		IF CalcolaFormingRT[IdxLista] AND NOT CalcolaFormingRT2[IdxLista] AND ActualPickingListFromHMI[IdxLista].State = 1   THEN //###############################  If  Principal calculos formaciones bendel y cabaleta
				 		//Para quitar
		Control1 := control1 +1 ;
			IF TFCalcoloFormaturaRT[IdxLista].CalcolaFormaturaDone THEN
				CalcolaFormaturaTrig2 := TRUE;	  
			END_IF
			IF NOT CalcolaFormaturaTrig2 AND NOT Formacion_bandelCalOk[idxForm]  THEN//11111111111111111
			///////////////////////////
				//CalcolaFormaturaTrig2 := TRUE;
				TFCalcoloFormaturaRT[IdxLista].PulisciMemoria 	:= TRUE;
				IF TFCalcoloFormaturaRT[IdxLista].PulisciMemoriaDone THEN		
					FOR i:= 1 TO MAXFORMINGSLAB DO
						IF i <= 40 THEN
						//IF i <= HMI_Forming_NumeroElementiDaDepositare THEN
							TFCalcoloFormaturaRT[IdxLista].TipoElementoDep[i] := LASTRA;//Settiamo tutte lastre!!
						ELSE
							TFCalcoloFormaturaRT[IdxLista].TipoElementoDep[i] := TERMINATORE;//Settiamo il resto come terminatore
						END_IF
					END_FOR
					TFCalcoloFormaturaRT[IdxLista].Materiale[e_Tipo_Elemento_Da_Lavorare.LASTRA].XDim		:= RequestPickingListFromHMI[IdxLista].SlabDimension.XDim; 
					TFCalcoloFormaturaRT[IdxLista].Materiale[e_Tipo_Elemento_Da_Lavorare.LASTRA].YDim		:= RequestPickingListFromHMI[IdxLista].SlabDimension.YDim; 
					TFCalcoloFormaturaRT[IdxLista].Materiale[e_Tipo_Elemento_Da_Lavorare.LASTRA].ZDim		:= RequestPickingListFromHMI[IdxLista].SlabDimension.ZDim; 
					TFCalcoloFormaturaRT[IdxLista].Supporto.Code											:= RequestPickingListFromHMI[IdxLista].SupportVertBundle.Code;
					TFCalcoloFormaturaRT[IdxLista].Supporto.XDim											:= RequestPickingListFromHMI[IdxLista].SupportVertBundle.XDim;
					TFCalcoloFormaturaRT[IdxLista].Supporto.YDim											:= RequestPickingListFromHMI[IdxLista].SupportVertBundle.YDim*2;
					TFCalcoloFormaturaRT[IdxLista].Supporto.ZDim				:= RequestPickingListFromHMI[IdxLista].SupportVertBundle.ZDim;
					TFCalcoloFormaturaRT[IdxLista].Supporto.TipoPianoAppoggio 	:= 1;
					TFCalcoloFormaturaRT[IdxLista].Supporto.AltezzaDenteRitenuta:= 15;
					TFCalcoloFormaturaRT[IdxLista].Supporto.ZDim_Ext1        	:= TFCalcoloFormaturaRT[IdxLista].Supporto.ZDim + TFCalcoloFormaturaRT[IdxLista].Supporto.AltezzaDenteRitenuta;
					TFCalcoloFormaturaRT[IdxLista].Supporto.DimBaseUtile		:= RequestPickingListFromHMI[IdxLista].SupportVertBundle.DimBaseUtile;
					TFCalcoloFormaturaRT[IdxLista].Supporto.DimVertice 			:= RequestPickingListFromHMI[IdxLista].SupportVertBundle.DimVertice*2;
					TFCalcoloFormaturaRT[IdxLista].Supporto.HMAX 				:= RequestPickingListFromHMI[IdxLista].SupportVertBundle.HMAX;
					TFCalcoloFormaturaRT[IdxLista].Supporto.Tipologia 			:= BUNDLE;
					TFCalcoloFormaturaRT[IdxLista].Supporto.LatoDeposito 		:= 180;
					TFCalcoloFormaturaRT[IdxLista].TipoOrdinamento				:= 4;	//Ordinamento di deposito, prima un lato poi l'altro
					TFCalcoloFormaturaRT[IdxLista].CalcolaFormatura 			:= TRUE;//Lancio esecuzione dei calcoli
					MEMSET(ADR(FormaturaBundleRT[IdxLista]),0,SIZEOF(FormaturaBundleRT[IdxLista]));	//Pulisco la memoria di destinazione
					TFCalcoloFormaturaRT[IdxLista].PulisciMemoria := FALSE;
				END_IF
			ELSIF (TFCalcoloFormaturaRT[IdxLista].CalcolaFormaturaDone OR TFCalcoloFormaturaRT[IdxLista].Errore > 0) AND CalcolaFormaturaTrig2 THEN
				CalcolaFormaturaTrig2 := FALSE;
				TFCalcoloFormaturaRT[IdxLista].CalcolaFormatura := FALSE;
				TFFormacionBandelCalculada := TFCalcoloFormaturaRT[IdxLista]; 
				FormaturaBundleRT[IdxLista] := TFCalcoloFormaturaRT[IdxLista].FormingSlab;
				IF TFCalcoloFormaturaRT[IdxLista].Errore = 0 THEN
					CalcolaFormaturaTrig2 			:= FALSE;
					CalcolaFormingRT[IdxLista] 		:= FALSE;
					CalcolaFormingRT2[IdxLista]		:= TRUE;
					Formacion_bandelCalOk[idxForm] 			:= TRUE ;
				ELSE
					CalcolaFormingRT[IdxLista] 		:= TRUE;
					CalcolaFormaturaTrig2 			:= FALSE;
				END_IF
			END_IF
		//##############################Inicio##############################################		 
		//#########################Calculo cavaleta##########################################
		ELSIF CalcolaFormingRT2[IdxLista] AND NOT CalcolaFormingRT[IdxLista] AND ActualPickingListFromHMI[IdxLista].State = 1  THEN 
			IF NOT CalcolaFormaturaTrig2 AND NOT Formacion_FrameCalOk[idxForm] THEN
			///////////////////////////
				TFCalcoloFormaturaRT[IdxLista].PulisciMemoria 	:= TRUE;	  
				
					
				//TFCalcoloFormaturaRT[IdxLista].PulisciMemoria 	:= TRUE;
				IF TFCalcoloFormaturaRT[IdxLista].PulisciMemoriaDone THEN
					CalcolaFormaturaTrig2 := TRUE;		
					FOR i:= 1 TO MAXFORMINGSLAB DO
						//IF i <= 10  THEN
						IF i <= 40 THEN
						//IF i <= HMI_Forming_NumeroElementiDaDepositare  THEN
							TFCalcoloFormaturaRT[IdxLista].TipoElementoDep[i] := LASTRA;//Settiamo tutte lastre!!
						ELSE
							TFCalcoloFormaturaRT[IdxLista].TipoElementoDep[i] := TERMINATORE;//Settiamo il resto come terminatore
						END_IF
					END_FOR
					TFCalcoloFormaturaRT[IdxLista].Materiale[e_Tipo_Elemento_Da_Lavorare.LASTRA].XDim		:= RequestPickingListFromHMI[IdxLista].SlabDimension.XDim; 
					TFCalcoloFormaturaRT[IdxLista].Materiale[e_Tipo_Elemento_Da_Lavorare.LASTRA].YDim		:= RequestPickingListFromHMI[IdxLista].SlabDimension.YDim; 
					TFCalcoloFormaturaRT[IdxLista].Materiale[e_Tipo_Elemento_Da_Lavorare.LASTRA].ZDim		:= RequestPickingListFromHMI[IdxLista].SlabDimension.ZDim; 
					TFCalcoloFormaturaRT[IdxLista].HabiCalTodasCordenadas := true ;
					TFCalcoloFormaturaRT[IdxLista].Supporto.Code											:= RequestPickingListFromHMI[IdxLista].SupportVertCav.Code;
					TFCalcoloFormaturaRT[IdxLista].Supporto.XDim											:= RequestPickingListFromHMI[IdxLista].SupportVertCav.XDim;
					TFCalcoloFormaturaRT[IdxLista].Supporto.YDim											:= RequestPickingListFromHMI[IdxLista].SupportVertCav.YDim(**2*);
					TFCalcoloFormaturaRT[IdxLista].Supporto.ZDim				:= RequestPickingListFromHMI[IdxLista].SupportVertCav.ZDim;
					TFCalcoloFormaturaRT[IdxLista].Supporto.TipoPianoAppoggio 	:= 1;
					TFCalcoloFormaturaRT[IdxLista].Supporto.AltezzaDenteRitenuta:= 13;
					TFCalcoloFormaturaRT[IdxLista].Supporto.ZDim_Ext1        	:= TFCalcoloFormaturaRT[IdxLista].Supporto.ZDim + TFCalcoloFormaturaRT[IdxLista].Supporto.AltezzaDenteRitenuta;
					TFCalcoloFormaturaRT[IdxLista].Supporto.DimBaseUtile		:= RequestPickingListFromHMI[IdxLista].SupportVertCav.DimBaseUtile;
					TFCalcoloFormaturaRT[IdxLista].Supporto.DimVertice 			:= RequestPickingListFromHMI[IdxLista].SupportVertCav.DimVertice(**2*);
					TFCalcoloFormaturaRT[IdxLista].Supporto.HMAX 				:= RequestPickingListFromHMI[IdxLista].SupportVertCav.HMAX;
					TFCalcoloFormaturaRT[IdxLista].Supporto.Tipologia 			:= CAVALLETTO;
					TFCalcoloFormaturaRT[IdxLista].Supporto.LatoDeposito 		:= 0;
					TFCalcoloFormaturaRT[IdxLista].TipoOrdinamento				:= 1;	//Ordinamento di deposito, prima un lato poi l'altro
					TFCalcoloFormaturaRT[IdxLista].CalcolaFormatura 			:= TRUE;//Lancio esecuzione dei calcoli
					MEMSET(ADR(FormaturaAFRAMERT[IdxLista]),0,SIZEOF(FormaturaAFRAMERT[IdxLista]));	//Pulisco la memoria di destinazione
					TFCalcoloFormaturaRT[IdxLista].PulisciMemoria := FALSE;
				END_IF
			ELSIF (TFCalcoloFormaturaRT[IdxLista].CalcolaFormaturaDone OR TFCalcoloFormaturaRT[IdxLista].Errore > 0) AND CalcolaFormaturaTrig2 THEN
				CalcolaFormaturaTrig2 		:= FALSE;
				TFCalcoloFormaturaRT[IdxLista].CalcolaFormatura := FALSE;
				TFFormacionCavalleteCalculada := TFCalcoloFormaturaRT[IdxLista] ;
				FormaturaAFRAMERT[IdxLista] := TFCalcoloFormaturaRT[IdxLista].FormingSlab;
				
				//CalcolaFormingRT[IdxLista] := TRUE ; // modificacion probar
				IF TFCalcoloFormaturaRT[IdxLista].Errore = 0 THEN
					CalcolaFormaturaTrig2 		:= FALSE;
					CalcolaFormingRT[IdxLista] 	:= TRUE;
					CalcolaFormingRT2[IdxLista]	:= FALSE;
					Formacion_FrameCalOk[idxForm] 		:= TRUE ;
				ELSE
					//CalcolaFormingRT[IdxLista] := TRUE; // original	  
					CalcolaFormingRT2[IdxLista] := TRUE;
				//##############################Fin ##############################################		 
				//#########################Calculo cavaleta##########################################
				END_IF
			END_IF
				  
		END_IF //###############################  If  Principal calculos formaciones bendel y cabaleta
	
	TFCalcoloFormaturaRT[IdxLista]();
END_FOR	 
	 

	HMI_WorkAreaDataPicking_1_8 := ActualPickingListFromHMI[1].State >= 1;//Ordine postazioni 1..8 in lavoro
		 
	HMI_WorkAreaDataPicking_1_4 := (ActualPickingListFromHMI[2].State >= 1);//Ordine postazioni 1..4 in lavoro
	HMI_WorkAreaDataPicking_5_8 := (ActualPickingListFromHMI[3].State >= 1);//Ordine postazioni 5..8 in lavoro

//FOR IdxLista := 1 TO 3 DO
//	CASE IdxLista OF	 
//		1: Iforstart := 1; Iforend := MAXAREAPRESENT;
//		2: Iforstart := 1; Iforend := 4;
//		3: Iforstart := 5; Iforend := MAXAREAPRESENT;
//	END_CASE		 		   
//	FOR i:= Iforstart TO Iforend DO	
//		IF NumeroPezziPresentiPostazioneStart[i] = 0 AND WorkAreaState[i].P > 1 THEN
//			NumeroPezziPresentiPostazioneStart[i] := TO_UINT(WorkAreaState[i].P);
//		END_IF
//	
//		IF NOT HMI_WorkAreaDataPicking[i].Destinazione THEN
//			IF HMI_WorkAreaDataPicking[i].NumElementiDaLavorare > 0 THEN
//				//IF HMI_WorkAreaDataPicking[i].NumElementiDaLavorare >= TO_UINT(WorkAreaState[i].P)-1 THEN
//				//	HMI_NumeroLastreRimanentiOrdineAttuale[i] := HMI_WorkAreaDataPicking[i].NumElementiDaLavorare - TO_UINT(WorkAreaState[i].P);
//				//ELSE
//				//	HMI_NumeroLastreRimanentiOrdineAttuale[i] := 0;
//				//END_IF
//				IF HMI_WorkAreaDataPicking[i].NumElementiDaLavorare - (TO_UINT(WorkAreaState[i].P) - NumeroPezziPresentiPostazioneStart[i]) > 0 THEN
//					HMI_NumeroLastreRimanentiOrdineAttuale[i] := MIN(HMI_WorkAreaDataPicking[i].NumElementiDaLavorare,HMI_WorkAreaDataPicking[i].NumElementiDaLavorare - 
//																(NumeroPezziPresentiPostazioneStart[i] - TO_UINT(WorkAreaState[i].P)));
//				ELSE
//					HMI_NumeroLastreRimanentiOrdineAttuale[i] := 0;
//				END_IF
//			ELSE
//				HMI_NumeroLastreRimanentiOrdineAttuale[i] := 0;
//			END_IF
//		ELSE
//			IF NumeroPezziPresentiPostazioneStart[i] <= (TO_UINT(WorkAreaState[i].P)) AND NumeroPezziPresentiPostazioneStart[i]>0 THEN
//				HMI_NumeroLastreRimanentiOrdineAttuale[i] := TO_UINT(WorkAreaState[i].P) - NumeroPezziPresentiPostazioneStart[i]+1;
//			ELSE
//				HMI_NumeroLastreRimanentiOrdineAttuale[i] := 0;
//			END_IF
//		END_IF
//		IF (WorkAreaProductionList[i].Stato = e_Stato_ListaDiProduzione.LISTA_PROD_IN_ESECUZIONE OR WorkAreaProductionList[i].Stato = e_Stato_ListaDiProduzione.LISTA_PROD_ESEGUITA) AND WorkAreaState[i].P > 1 THEN
//			HMI_NumeroLastreDepOrdineAttuale[IdxLista] := TO_UINT(WorkAreaState[i].P-1);
//			IF NumeroPezziPresentiPostazioneStart[i] < (TO_UINT(WorkAreaState[i].P)) AND NumeroPezziPresentiPostazioneStart[i]>0 THEN
//				HMI_NumeroLastreDepOrdineAttuale[IdxLista] := TO_UINT(WorkAreaState[i].P) - NumeroPezziPresentiPostazioneStart[i] +1;
//			ELSE
//				HMI_NumeroLastreDepOrdineAttuale[IdxLista] := 0;
//			END_IF
//		END_IF	
//	END_FOR		  
//END_FOR			   
					
						 
							  
								   
{endregion}
END_ACTION

ACTION _11_CalcolaListaProduzioneNew:
{region "Gestione zona GLOBALE - Postazioni da 1 a 8"}


//#############################################################################################################



	  
	  

FOR LoopLista := 1 TO 3 DO
	IdxLista := LoopLista;		 
	 // IdxLista := 2;		  
	CASE IdxLista OF	 
		1: Iforstart := 1; Iforend := MAXAREAPRESENT;
		2: Iforstart := 1; Iforend := 4;
		3: Iforstart := 5; Iforend := MAXAREAPRESENT;
	END_CASE	 
IF MachinePalletizer_TF.IN.Mode.Man AND
		(MachinePalletizer_TF.CmdExe.Code = CmdNOP OR MachinePalletizer_TF.CmdExe.Code = CmdMAN) THEN
			 
				  
					   
							
{region "Reset Litas"}
//--------------------------------------------------------
			//AZZERAMENTO (Reset) lista di picking	
//--------------------------------------------------------		 
			IF Cmd_AzzeraLista[IdxLista] THEN
				IF Prueva AND FALSE THEN
					MissionClr := ADR(Mission) ;
	 				MEMSET(destAddr := ADR(MissionClr^),fillByte := 0 , n := SIZEOF(MissionClr^));
				END_IF
					ClrEstructura := ADR(PosCavalleteOrdenPikin) ;
					MEMSET(destAddr := ADR(ClrEstructura^),fillByte := 0 , n := SIZEOF(ClrEstructura^));	  
					NuEstacionesPiking := 0 ;	  
					NuEstacionPiking   := 0 ;
					NuPosGuiroPiking := 0;
					PosFinOrdenPikingCaballete := 0 ;
					
					MultiplesCavalletesReceta := FALSE ;
					CoordenadaPasillo0_Y := 0 ;
					CoordenadaPasillo180_Y := 0 ;
					
				
				//FOR i:= 1 TO 3 DO
						//CalcolaFormingRT2[i] := FALSE ;
					CalcolaFormingRT[IdxLista] := FALSE ;
					CalcolaFormingRT2[IdxLista] := FALSE ;	 
						//#Añadido 4_7_2025########################
					Formacion_bandelCalOk[IdxLista]			:= FALSE ;
					Formacion_FrameCalOk[IdxLista]			:= FALSE ;
					Formacion_De_listaOk[IdxLista]			:= FALSE ;
					FormaturaAFRAMERT[IdxLista]		   	:=	FormingEmpty;
					FormaturaBundleRT[IdxLista]	 		:=	FormingEmpty;
							  
					MEMSET(destAddr := ADR(TFFormacionBandelCalculada),fillByte := 0 , n := SIZEOF(TFFormacionBandelCalculada));
					MEMSET(destAddr := ADR(TFFormacionCavalleteCalculada),fillByte := 0 , n := SIZEOF(TFFormacionCavalleteCalculada));
					MEMSET(destAddr := ADR(TFCalcoloFormaturaWA),fillByte := 0 , n := SIZEOF(TFCalcoloFormaturaWA));
					MEMSET(destAddr := ADR(HMI_Forming_FormaturaAttivataWa),fillByte := 0 , n := SIZEOF(HMI_Forming_FormaturaAttivataWa));
				
							MEMSET(destAddr := ADR(HMi_DimensionesPiezasWorkAreaDeposito),fillByte := 0 , n := SIZEOF(HMi_DimensionesPiezasWorkAreaDeposito));			  
				
				
					
					FormacionesCalculadas := FALSE ;
					FormacionPikingCalculada := FALSE ;
				(*	FOR i:= Iforstart TO Iforend DO	
						TFCalcoloFormaturaWA[i].PulisciMemoria := TRUE ;
		  			END_FOR *)
				//Añadido 4_7_2025##########################
						
				// END_FOR
				ActualPickingListFromHMI[IdxLista].State := e_StatoWorkOrder.NON_ESEGUITO;
				HMI_NumeroLastreDepOrdineAttuale[IdxLista] := 0; 
				//Disattivazione formatura
				Forming[1] := FormingEmpty;	//Pulisco la formatura selezionata e di consegenza la disattivo
				Forming[2] := FormingEmpty;	//Pulisco la formatura selezionata e di consegenza la disattivo
				Forming[3] := FormingEmpty;	//Pulisco la formatura selezionata e di consegenza la disattivo
				Forming[4] := FormingEmpty;	//Pulisco la formatura selezionata e di consegenza la disattivo
				ActualPickingListFromHMI[IdxLista].State := e_StatoWorkOrder.NON_ESEGUITO;
				Cmd_AttivaLista[IdxLista] := FALSE;
				HMI_Forming_NumeroElementiDaDepositare := 0;
 				RequestPickingListFromHMI[IdxLista].SlabNumber :=0;
	 
				//Azzero le liste per le postazioni dove non avviene la pallettizzazione
				FOR i:= Iforstart TO Iforend DO	
					TFClearWorkAreaArray(ADR(Workarea),ADR(WorkAreaState),k:=i);
					HMI_WorkAreaDataPicking[i].Destinazione := FALSE;
					HMI_WorkAreaDataPicking[i].NumElementiDaLavorare := 0;
					WorkAreaState[i].P 			:= 1;
					WorkAreaProductionList[i] 	:= ListaEmpty;
					WorkAreaOffset[i].Y 		:= 0;
					//HMI_NumeroPezziPresentiPostazione[i] 	:= 0; // Quitado Para No resetear posiciones
					NumeroPezziPresentiPostazioneStart[i] 	:= 0;
					WorkAreaProductionList[i].Stato 		:= e_Stato_ListaDiProduzione.LISTA_PROD_ASSENTE;	 
				END_FOR			  
				ActualPickingListFromHMI[IdxLista].SlabNumber 		  			:= 0;
				ActualPickingListFromHMI[IdxLista].SlabDimension.XDim 			:= 0;
				ActualPickingListFromHMI[IdxLista].SlabDimension.YDim 			:= 0;
				ActualPickingListFromHMI[IdxLista].SlabDimension.ZDim 			:= 0;
				ActualPickingListFromHMI[IdxLista].SupportPianoLegno 			:= SupportDataEmpty;
				ActualPickingListFromHMI[IdxLista].SupportPianoFerro 			:= SupportDataEmpty;
				ActualPickingListFromHMI[IdxLista].SupportVertBundle 			:= SupportDataEmpty;
				ActualPickingListFromHMI[IdxLista].SupportVertCav 			 	:= SupportDataEmpty;
				
				HMI_ErroreCalcoloLista 		:= 0;
				Cmd_CalcolaLista[IdxLista] 	:= FALSE;
				HMI_Forming_Attivazione[IdxLista] 	:= FALSE;//attivo nuova formatura
				Cmd_AzzeraLista[IdxLista] := FALSE;
				//Ack 
				//IF HMI_ErrAckCalcolaFormatura THEN
					HMI_Forming_ErroreCalcoli := 0;
					HMI_ErrAckCalcolaFormatura := FALSE;
					FOR i:= 1 TO MAXFORMING DO
						HMI_ConfermaAttivazioneFormatura[i] := FALSE;
						HMI_Forming_FormaturaAttivata[i] := FALSE;
					END_FOR
				//END_IF
				CalcolaFormaturaTrig := FALSE;
			END_IF

{endregion}

//--------------------------------------------------------
		// COMANDO ATTIVAZIONE  lista di picking	
//--------------------------------------------------------		 		  
			//Se non ho una Destinazione impostata, Num.pezzi impostato, o Num.pezzi richiesto...
			//	Resetto il comando		
					IF Cmd_AttivaLista[1] = TRUE  THEN
							FOR uu := Iforstart TO Iforend DO
							 	IF	HMI_WorkAreaDataPicking[uu].Typology = CAVALLETTO THEN 
									CASE HMI_WorkAreaDataPicking[uu].TipoTrabajoLado_Cavallete OF 
	 									0:
											HMI_NumeroPezziPresentiPostazione[uu] := HMI_NumeroPezziPresentiCavallete[uu].HMI_NumeroPezziPresentiPostazione_A_Cavaleto +
												 HMI_NumeroPezziPresentiCavallete[uu].HMI_NumeroPezziPresentiPostazione_B_Cavaleto ;
										1:
											HMI_NumeroPezziPresentiPostazione[uu] := HMI_NumeroPezziPresentiCavallete[uu].HMI_NumeroPezziPresentiPostazione_A_Cavaleto ;									 ;
											 
										2:	
		   									HMI_NumeroPezziPresentiPostazione[uu] := HMI_NumeroPezziPresentiCavallete[uu].HMI_NumeroPezziPresentiPostazione_B_Cavaleto ;
												 
									END_CASE
								END_IF 	 
							END_FOR
								  
						IF 	(HMI_WorkAreaDataPicking[1].Destinazione =0 AND 
							HMI_WorkAreaDataPicking[2].Destinazione =0 AND
							HMI_WorkAreaDataPicking[3].Destinazione =0 AND 
							HMI_WorkAreaDataPicking[4].Destinazione =0 AND	 
							HMI_WorkAreaDataPicking[5].Destinazione =0 AND 
							HMI_WorkAreaDataPicking[6].Destinazione =0 AND
							HMI_WorkAreaDataPicking[7].Destinazione =0 AND 
							HMI_WorkAreaDataPicking[8].Destinazione =0)							 
							OR
							(HMI_NumeroPezziPresentiPostazione[1] =0 AND 
							HMI_NumeroPezziPresentiPostazione[2] =0 AND
							HMI_NumeroPezziPresentiPostazione[3] =0 AND 
							HMI_NumeroPezziPresentiPostazione[4] =0 AND
							HMI_NumeroPezziPresentiPostazione[5] =0 AND 
	 						HMI_NumeroPezziPresentiPostazione[6] =0 AND
							HMI_NumeroPezziPresentiPostazione[7] =0 AND 
							HMI_NumeroPezziPresentiPostazione[8] =0)
							OR	 	 
							RequestPickingListFromHMI[1].SlabNumber = 0	 
						THEN
							Cmd_AttivaLista[1] := FALSE;
						 END_IF
					END_IF		  
					IF Cmd_AttivaLista[2] = TRUE  THEN
							FOR uu := Iforstart TO Iforend DO
							 	IF	HMI_WorkAreaDataPicking[uu].Typology = CAVALLETTO THEN 
									CASE HMI_WorkAreaDataPicking[uu].TipoTrabajoLado_Cavallete OF 
	 									0:
											HMI_NumeroPezziPresentiPostazione[uu] := HMI_NumeroPezziPresentiCavallete[uu].HMI_NumeroPezziPresentiPostazione_A_Cavaleto +
												 HMI_NumeroPezziPresentiCavallete[uu].HMI_NumeroPezziPresentiPostazione_B_Cavaleto ;
										1:
											HMI_NumeroPezziPresentiPostazione[uu] := HMI_NumeroPezziPresentiCavallete[uu].HMI_NumeroPezziPresentiPostazione_A_Cavaleto ;									 ;
											 
										2:	
		   									HMI_NumeroPezziPresentiPostazione[uu] := HMI_NumeroPezziPresentiCavallete[uu].HMI_NumeroPezziPresentiPostazione_B_Cavaleto ;
												 
									END_CASE
								END_IF 	 
							END_FOR
						IF 	(HMI_WorkAreaDataPicking[1].Destinazione =0 AND 
							HMI_WorkAreaDataPicking[2].Destinazione =0 AND
							HMI_WorkAreaDataPicking[3].Destinazione =0 AND 
							HMI_WorkAreaDataPicking[4].Destinazione =0)
							OR
							(HMI_NumeroPezziPresentiPostazione[1] =0 AND 
							HMI_NumeroPezziPresentiPostazione[2] =0 AND
							HMI_NumeroPezziPresentiPostazione[3] =0 AND 
							HMI_NumeroPezziPresentiPostazione[4] =0)
							OR	 
							RequestPickingListFromHMI[2].SlabNumber = 0	 	 
						THEN
							Cmd_AttivaLista[2] := FALSE;
						 END_IF
					END_IF		
					IF Cmd_AttivaLista[3] = TRUE  THEN
							FOR uu := Iforstart TO Iforend DO
							 	IF	HMI_WorkAreaDataPicking[uu].Typology = CAVALLETTO THEN 
									CASE HMI_WorkAreaDataPicking[uu].TipoTrabajoLado_Cavallete OF 
	 									0:
											HMI_NumeroPezziPresentiPostazione[uu] := HMI_NumeroPezziPresentiCavallete[uu].HMI_NumeroPezziPresentiPostazione_A_Cavaleto +
												 HMI_NumeroPezziPresentiCavallete[uu].HMI_NumeroPezziPresentiPostazione_B_Cavaleto ;
										1:
											HMI_NumeroPezziPresentiPostazione[uu] := HMI_NumeroPezziPresentiCavallete[uu].HMI_NumeroPezziPresentiPostazione_A_Cavaleto ;									 ;
											 
										2:	
		   									HMI_NumeroPezziPresentiPostazione[uu] := HMI_NumeroPezziPresentiCavallete[uu].HMI_NumeroPezziPresentiPostazione_B_Cavaleto ;
												 
									END_CASE
								END_IF 	 
							END_FOR
						IF 	(HMI_WorkAreaDataPicking[5].Destinazione =0 AND 
							HMI_WorkAreaDataPicking[6].Destinazione =0 AND
							HMI_WorkAreaDataPicking[7].Destinazione =0 AND 
							HMI_WorkAreaDataPicking[8].Destinazione =0)
							OR
							(HMI_NumeroPezziPresentiPostazione[5] =0 AND 
							HMI_NumeroPezziPresentiPostazione[6] =0 AND
							HMI_NumeroPezziPresentiPostazione[7] =0 AND 
							HMI_NumeroPezziPresentiPostazione[8] =0)
							OR	 	 
							RequestPickingListFromHMI[3].SlabNumber = 0	 	 
						THEN
							Cmd_AttivaLista[3] := FALSE;
						 END_IF
					END_IF		
{Region "Prmer Bucle cuenta las piezas a coger y rellena el workareastate Con el Tipo Palet"}

			// COMANDO ATTIVAZIONE  lista di picking	
		    IF Cmd_AttivaLista[IdxLista] AND ActualPickingListFromHMI[IdxLista].State <> e_StatoWorkOrder.IN_ESECUZIONE THEN
				ElementiDaDepositare[IdxLista]   :=0;
				HMI_ErroreCalcoloLista := 0;
				HMI_NumeroLastreDepOrdineAttuale[IdxLista] := 0;
				FOR i:= Iforstart TO Iforend DO	
					//HMI_WorkAreaDataPicking[i].Destinazione := FALSE;
					//HMI_WorkAreaDataPicking[i].NumElementiDaLavorare := 0;
					WorkAreaState[i].P := 1;
					WorkAreaProductionList[i] := ListaEmpty;
				END_FOR	 
				
				FOR i:= Iforstart TO Iforend DO	
					IF NOT HMI_WorkAreaDataPicking[i].Destinazione THEN
						ElementiDaDepositare[IdxLista] := ElementiDaDepositare[IdxLista] + HMI_WorkAreaDataPicking[i].NumElementiDaLavorare;
						WorkAreaState[i].P := HMI_WorkAreaDataPicking[i].NumElementiDaLavorare +1;
					//#####################################################################################
							FOR InPiezasPos := 1 TO HMI_NumeroPezziPresentiPostazione[i] + 1 DO
								WorkAreaProductionList[i].PElementList[InPiezasPos].PElement.SlabDimension :=
																	 RequestPickingListFromHMIWorkArea[i].SlabDimension ;
								WorkAreaProductionList[i].PElementList[InPiezasPos].PElement.Typology := LASTRA ;
											   
							END_FOR
					//#################################################################################################	
						CASE HMI_WorkAreaDataPicking[i].Typology OF
							LEGNO_PIANO,TELAIO_PIANO:
								WorkareaState[i].Supporto.Tipologia := e_Tipo_Pallet.CASSA_STANDARD;
							A_FRAME_VERT:	
								WorkareaState[i].Supporto.Tipologia := e_Tipo_Pallet.CAVALLETTO;
								
							IF HMI_WorkAreaDataPicking[i].NumElementiDaLavorare > 0 THEN 
								NuEstacionesPiking := NuEstacionesPiking + 1 ;	
								PosCavalleteOrdenPikin[i]	:=  e_Tipo_Pallet.CAVALLETTO;  
							END_IF
							BUNDLE_VERT:
								WorkareaState[i].Supporto.Tipologia := e_Tipo_Pallet.BUNDLE;	
							
						 ELSE
								WorkareaState[i].Supporto.Tipologia := e_Tipo_Pallet.CASSA_STANDARD;		   
						 END_CASE
					ELSE
						NumPostazioneDeposito := i; NuEstacionPiking := i;
						
						HMI_WorkAreaDataPicking[NumPostazioneDeposito].NumElementiDaLavorare := RequestPickingListFromHMI[IdxLista].SlabNumber;
						CASE HMI_WorkAreaDataPicking[i].Typology OF
							LEGNO_PIANO,TELAIO_PIANO:
								WorkareaState[i].Supporto.Tipologia := e_Tipo_Pallet.CASSA_STANDARD;
							A_FRAME_VERT:	
								WorkareaState[i].Supporto.Tipologia := e_Tipo_Pallet.CAVALLETTO;
								NuEstacionesPiking := NuEstacionesPiking + 1 ;	
								PosCavalleteOrdenPikin[i]	:=  e_Tipo_Pallet.CAVALLETTO;  	 
							BUNDLE_VERT:
								WorkareaState[i].Supporto.Tipologia := e_Tipo_Pallet.BUNDLE;	
								
							
						 ELSE
								WorkareaState[i].Supporto.Tipologia := e_Tipo_Pallet.CASSA_STANDARD;		   
						 END_CASE
					END_IF

		  
//HMI_NumeroPezziPresentiPostazione[i] := WorkAreaState[i].P -1; //NB:cancellato xckè alla attivazione azzerava il num.pezzi presenti sulle postazioni di prelievo
				END_FOR
	
				IF ElementiDaDepositare[IdxLista] <= HMI_WorkAreaDataPicking[NumPostazioneDeposito].NumElementiDaLavorare THEN
					ActualPickingListFromHMI[IdxLista] 			:= RequestPickingListFromHMI[IdxLista];
					ActualPickingListFromHMI[IdxLista].State 	:= e_StatoWorkOrder.DA_ESEGUIRE;

				ELSE
					HMI_ErroreCalcoloLista := 1;
				END_IF
				Cmd_AttivaLista[IdxLista] 				:= FALSE;
				 
			ELSE
				Cmd_AttivaLista[IdxLista] 				:= FALSE;
				 
			END_IF
{endregion}	

{region "Cotas posicione de trabajo"}

//--------------------------------------------------------------------				
//////// attivazione lista di picking : StatoWorkOrder.DA_ESEGUIRE ///
//--------------------------------------------------------------------				
			IF ActualPickingListFromHMI[IdxLista].State = e_StatoWorkOrder.DA_ESEGUIRE  THEN
				ListaInEsecuzione[IdxLista] := FALSE;
				NumeroListaInEsecuzione := 0;
			
				(* Inserimento sequenza di prelievo dalle postazioni in base al quello che l'operatore ha editato da HMI*)
				ElementiDaDepositare[IdxLista] := 0;
				ElementiElaborati[IdxLista]    := 1;
				NumPostazioneDeposito := 0;
				//FOR i:= 1 TO MAXAREAPRESENT DO
				//	WorkAreaState[i].P := 1;
				//END_FOR		
				
				FOR i:= Iforstart TO Iforend DO//---------- For 1 HMI_WorkAreaDataPicking[i].Destinazione 
					IF HMI_WorkAreaDataPicking[i].Destinazione THEN  //-------> Palet destino
						NumPostazioneDeposito := i;
						Numero_Piezas_estacionPikin := HMI_NumeroPezziPresentiPostazione[NumPostazioneDeposito] +1 ;
						Numero_piezas_CaballeteEstacionPiking.HMI_NumeroPezziPresentiPostazione_A_Cavaleto := HMI_NumeroPezziPresentiCavallete[NumPostazioneDeposito].HMI_NumeroPezziPresentiPostazione_A_Cavaleto +1 ;
						Numero_piezas_CaballeteEstacionPiking.HMI_NumeroPezziPresentiPostazione_B_Cavaleto := HMI_NumeroPezziPresentiCavallete[NumPostazioneDeposito].HMI_NumeroPezziPresentiPostazione_B_Cavaleto +1 ;
						HMI_WorkAreaDataPicking[NumPostazioneDeposito].NumElementiDaLavorare 	:= RequestPickingListFromHMI[IdxLista].SlabNumber;
						(*CASE HMI_WorkAreaDataPicking[i].Typology OF     // case Pricipal1*)		 
						CASE HMI_WorkAreaDataPicking[NumPostazioneDeposito].Typology OF     // case Pricipal1	
							(* Se ho un legno in piano *)	 
							LEGNO_PIANO:	
								//WorkAreaState[NumPostazioneDeposito].Supporto.Code 						:= ActualPickingListFromHMI[IdxLista].SupportPianoLegno.Code; 
								WorkAreaState[NumPostazioneDeposito].Supporto.Code 						:= RequestPickingListFromHMIWorkArea[i].SupportPianoLegno.Code; 	   
								//WorkAreaState[NumPostazioneDeposito].Supporto.AltezzaDenteRitenuta 		:= ActualPickingListFromHMI[IdxLista].SupportPianoLegno.DimBaseUtile;
								WorkAreaState[NumPostazioneDeposito].Supporto.AltezzaDenteRitenuta 		:= RequestPickingListFromHMIWorkArea[i].SupportPianoLegno.DimBaseUtile;
								//WorkAreaState[NumPostazioneDeposito].Supporto.DimVertice 				:= ActualPickingListFromHMI[IdxLista].SupportPianoLegno.DimVertice;
								WorkAreaState[NumPostazioneDeposito].Supporto.DimVertice 				:= RequestPickingListFromHMIWorkArea[i].SupportPianoLegno.DimVertice;			   
								//WorkAreaState[NumPostazioneDeposito].Supporto.HMAX 						:= ActualPickingListFromHMI[IdxLista].SupportPianoLegno.HMAX;
							   	WorkAreaState[NumPostazioneDeposito].Supporto.HMAX 						:= RequestPickingListFromHMIWorkArea[i].SupportPianoLegno.HMAX;
								//WorkAreaState[NumPostazioneDeposito].Supporto.Tipologia 				:= e_Tipo_Pallet.CASSA_STANDARD;//ActualPickingListFromHMI.Support.Tipologia;
								WorkAreaState[NumPostazioneDeposito].Supporto.Tipologia 				:= e_Tipo_Pallet.CASSA_STANDARD;//ActualPickingListFromHMI.Support.Tipologia;   
								//WorkAreaState[NumPostazioneDeposito].Supporto.XDim 						:= ActualPickingListFromHMI[IdxLista].SupportPianoLegno.XDim;
								WorkAreaState[NumPostazioneDeposito].Supporto.XDim 						:= RequestPickingListFromHMIWorkArea[i].SupportPianoLegno.XDim;
								//WorkAreaState[NumPostazioneDeposito].Supporto.YDim 						:= ActualPickingListFromHMI[IdxLista].SupportPianoLegno.YDim;
								WorkAreaState[NumPostazioneDeposito].Supporto.YDim 						:= RequestPickingListFromHMIWorkArea[i].SupportPianoLegno.YDim;
								//WorkAreaState[NumPostazioneDeposito].Supporto.ZDim 						:= ActualPickingListFromHMI[IdxLista].SupportPianoLegno.ZDim;
								WorkAreaState[NumPostazioneDeposito].Supporto.ZDim 						:= RequestPickingListFromHMIWorkArea[i].SupportPianoLegno.ZDim;
								WorkAreaOffset[NumPostazioneDeposito].Y 								:= OFFSET_POSTAZIONE_LEGNO + WorkAreaState[NumPostazioneDeposito].Supporto.XDim/2;//ATTENZIONE!!! per poter lavorare in centro con i supporti pari, questa misura è la distanza tra il riscontro bundle verticale e il centro postazione PARI
								
								WorkAreaProductionList[NumPostazioneDeposito].Support 				:= WorkAreaState[NumPostazioneDeposito].Supporto;
								
								FOR j:= Iforstart TO Iforend DO
									IF NOT HMI_WorkAreaDataPicking[j].Destinazione THEN
										IF HMI_WorkAreaDataPicking[j].NumElementiDaLavorare >= 1 THEN
											
											ElementiDaDepositare[IdxLista] := ElementiElaborati[IdxLista] + HMI_WorkAreaDataPicking[j].NumElementiDaLavorare;
											FOR k := ElementiElaborati[IdxLista] TO ElementiDaDepositare[IdxLista]-1 DO	
												WorkAreaProductionList[NumPostazioneDeposito].PElementList[k].WA_PRELIEVO := j;
												WorkAreaProductionList[NumPostazioneDeposito].PElementList[k].WA_DEPOSITO := i;	
												ElementiElaborati[IdxLista] := ElementiElaborati[IdxLista]+1; 
											END_FOR
												pr1 := 	Numero_Piezas_estacionPikin ;  
												pr2 := Numero_Piezas_estacionPikin  + HMI_WorkAreaDataPicking[j].NumElementiDaLavorare -1 ;				
											FOR ja := Numero_Piezas_estacionPikin  TO Numero_Piezas_estacionPikin  + HMI_WorkAreaDataPicking[j].NumElementiDaLavorare-1 DO
												// Se van Añadiendo los Diferentes Espesores de la receta del piking ######################################
												HMi_DimensionesPiezasWorkAreaDeposito[ja].Dim_Horizontal := RequestPickingListFromHMIWorkArea[j].SlabDimension ;
												//########################################################################################################		  
											END_FOR		  
												Numero_Piezas_estacionPikin := Numero_Piezas_estacionPikin +HMI_WorkAreaDataPicking[j].NumElementiDaLavorare; 	
											CASE HMI_WorkAreaDataPicking[j].Typology OF 
												(* Se ho una cassa pianale in legno *)
												LEGNO_PIANO:
													WorkAreaState[j].Supporto.Code 					:= RequestPickingListFromHMIWorkArea[j].SupportPianoLegno.Code;
													WorkAreaState[j].Supporto.DimBaseUtile		 	:= RequestPickingListFromHMIWorkArea[j].SupportPianoLegno.DimBaseUtile;
													WorkAreaState[j].Supporto.AltezzaDenteRitenuta 	:= RequestPickingListFromHMIWorkArea[j].SupportPianoLegno.ZDim+20;
													WorkAreaState[j].Supporto.DimVertice 			:= RequestPickingListFromHMIWorkArea[j].SupportPianoLegno.DimVertice;
													WorkAreaState[j].Supporto.HMAX 					:= RequestPickingListFromHMIWorkArea[j].SupportPianoLegno.HMAX;
													WorkAreaState[j].Supporto.Tipologia 			:= e_Tipo_Pallet.CASSA_STANDARD;//ActualPickingListFromHMI[1].Support.Tipologia;
													WorkAreaState[j].Supporto.XDim 					:= RequestPickingListFromHMIWorkArea[j].SupportPianoLegno.XDim;
													WorkAreaState[j].Supporto.YDim 					:= RequestPickingListFromHMIWorkArea[j].SupportPianoLegno.YDim;
													WorkAreaState[j].Supporto.ZDim 					:= RequestPickingListFromHMIWorkArea[j].SupportPianoLegno.ZDim;
													WorkAreaOffset[j].Y 							:= OFFSET_POSTAZIONE_LEGNO + WorkAreaState[j].Supporto.YDim/2;//ATTENZIONE!!! per poter lavorare in centro con i supporti pari, questa misura è la distanza tra il riscontro bundle verticale e il centro postazione PARI
													
																   
												(* Se ho una cassa pianale in ferro su supporto *)
												TELAIO_PIANO:
													WorkAreaState[j].Supporto.Code 					:= RequestPickingListFromHMIWorkArea[j].SupportPianoFerro.Code;
													WorkAreaState[j].Supporto.DimBaseUtile		 	:= RequestPickingListFromHMIWorkArea[j].SupportPianoFerro.DimBaseUtile;
													WorkAreaState[j].Supporto.AltezzaDenteRitenuta 	:= RequestPickingListFromHMIWorkArea[j].SupportPianoFerro.ZDim+20;
													WorkAreaState[j].Supporto.DimVertice 			:= RequestPickingListFromHMIWorkArea[j].SupportPianoFerro.DimVertice;
													WorkAreaState[j].Supporto.HMAX 					:= RequestPickingListFromHMIWorkArea[j].SupportPianoFerro.HMAX;
													WorkAreaState[j].Supporto.Tipologia 			:=  e_Tipo_Pallet.CASSA_STANDARD;//ActualPickingListFromHMI[1].Support.Tipologia;
													WorkAreaState[j].Supporto.XDim 					:= RequestPickingListFromHMIWorkArea[j].SupportPianoFerro.XDim;
													WorkAreaState[j].Supporto.YDim 					:= RequestPickingListFromHMIWorkArea[j].SupportPianoFerro.YDim;
													WorkAreaState[j].Supporto.ZDim 					:= RequestPickingListFromHMIWorkArea[j].SupportPianoFerro.ZDim;
													WorkAreaOffset[j].Y 							:= OFFSET_POSTAZIONE_TELAIO - WorkAreaState[j].Supporto.YDim/2;//ATTENZIONE!!! per poter lavorare in centro con i supporti pari, questa misura è la distanza tra il riscontro bundle verticale e il centro postazione PARI
												(* Se ho un bundle *)
												BUNDLE_VERT:
													//WorkAreaState[j].P := ElementiDaDepositare;
													WorkAreaState[j].Supporto.Code 					:= RequestPickingListFromHMIWorkArea[j].SupportVertBundle.Code;
													WorkAreaState[j].Supporto.DimBaseUtile		 	:= RequestPickingListFromHMIWorkArea[j].SupportVertBundle.DimBaseUtile;
													WorkAreaState[j].Supporto.AltezzaDenteRitenuta 	:= RequestPickingListFromHMIWorkArea[j].SupportVertBundle.ZDim+20;
													WorkAreaState[j].Supporto.DimVertice 			:= RequestPickingListFromHMIWorkArea[j].SupportVertBundle.DimVertice;
													WorkAreaState[j].Supporto.HMAX 					:= RequestPickingListFromHMIWorkArea[j].SupportVertBundle.HMAX;
													WorkAreaState[j].Supporto.Tipologia 			:= e_Tipo_Pallet.BUNDLE;//ActualPickingListFromHMI.SupportVert.Tipologia;
													WorkAreaState[j].Supporto.XDim 					:= RequestPickingListFromHMIWorkArea[j].SupportVertBundle.XDim;
													WorkAreaState[j].Supporto.YDim 					:= RequestPickingListFromHMIWorkArea[j].SupportVertBundle.YDim;
													WorkAreaState[j].Supporto.ZDim 					:= RequestPickingListFromHMIWorkArea[j].SupportVertBundle.ZDim;
													WorkAreaState[j].Supporto.ZDim_Ext1        		:= WorkAreaState[j].Supporto.ZDim + 20;
													WorkAreaState[j].Supporto.TipoPianoAppoggio 	:= 1;                      
													WorkAreaState[j].Supporto.AltezzaDenteRitenuta	:= 20; 
													WorkAreaState[j].Supporto.LatoDeposito 			:= 180;    
													WorkAreaOffset[j].Y 							:= 0 ;			
												(* Se ho un A_Frame *)	  
												A_FRAME_VERT:  						
													//WorkAreaState[j].P := ElementiDaDepositare;
													WorkAreaState[j].Supporto.Code 					:= ActualPickingListFromHMI[IdxLista].SupportVertCav.Code;
													WorkAreaState[j].Supporto.DimBaseUtile		 	:= RequestPickingListFromHMIWorkArea[j].SupportVertCav.DimBaseUtile;
													WorkAreaState[j].Supporto.AltezzaDenteRitenuta 	:= RequestPickingListFromHMIWorkArea[j].SupportVertCav.ZDim+20;
													WorkAreaState[j].Supporto.DimVertice 			:= RequestPickingListFromHMIWorkArea[j].SupportVertCav.DimVertice;
													WorkAreaState[j].Supporto.HMAX 					:= RequestPickingListFromHMIWorkArea[j].SupportVertCav.HMAX;
													WorkAreaState[j].Supporto.Tipologia 			:= CAVALLETTO;//ActualPickingListFromHMI.SupportVertCav.Tipologia;
													WorkAreaState[j].Supporto.XDim 					:= RequestPickingListFromHMIWorkArea[j].SupportVertCav.XDim;
													WorkAreaState[j].Supporto.YDim 					:= RequestPickingListFromHMIWorkArea[j].SupportVertCav.YDim;
													WorkAreaState[j].Supporto.ZDim 					:= RequestPickingListFromHMIWorkArea[j].SupportVertCav.ZDim;
													WorkAreaState[j].Supporto.ZDim_Ext1        		:= WorkAreaState[j].Supporto.ZDim + 20;	
													WorkAreaState[j].Supporto.TipoPianoAppoggio 	:= 1;                      
													WorkAreaState[j].Supporto.AltezzaDenteRitenuta	:= 15; 
													WorkAreaState[j].Supporto.TipoTrabajoLado_Cavallete := HMI_WorkAreaDataPicking[j].TipoTrabajoLado_Cavallete ; 	
													WorkAreaOffset[j].Y 							:= OFFSET_POSTAZIONE_LEGNO + WorkAreaState[j].Supporto.YDim/2;//ATTENZIONE!!! per poter lavorare in centro con i supporti pari, questa misura è la distanza tra il riscontro bundle verticale e il centro postazione PARI
											   		CoordenadaPasillo0_Y 							:= WorkArea[j].Y + WorkAreaOffset[j].Y  - Dimensioni_Pinza.Spessore - INGOMBRO_RISCONTRO_FRAME - WorkAreaState[j].Supporto.YDim /2 ;
													CoordenadaPasillo180_Y 							:= WorkArea[j].Y + WorkAreaState[j].Supporto.YDim /2 + WorkAreaOffset[j].Y  + Dimensioni_Pinza.Spessore + INGOMBRO_RISCONTRO_FRAME  ;	
											END_CASE	
											WorkAreaProductionList[j].Support := WorkAreaState[j].Supporto; 
										END_IF
									END_IF     
									TFClearApprendimento(ADR(WorkAreaState[j].Apprendimento));//Azzeramento apprendimento 
								END_FOR
								EXIT; 
							(* Se ho un telaio in piano *)	 
							TELAIO_PIANO:	
								
								WorkAreaState[NumPostazioneDeposito].Supporto.Code 						:= ActualPickingListFromHMI[IdxLista].SupportPianoFerro.Code;
								WorkAreaState[NumPostazioneDeposito].Supporto.AltezzaDenteRitenuta 		:= RequestPickingListFromHMIWorkArea[NumPostazioneDeposito].SupportPianoFerro.DimBaseUtile;
								WorkAreaState[NumPostazioneDeposito].Supporto.DimVertice 				:= RequestPickingListFromHMIWorkArea[NumPostazioneDeposito].SupportPianoFerro.DimVertice;
								WorkAreaState[NumPostazioneDeposito].Supporto.HMAX 						:= RequestPickingListFromHMIWorkArea[NumPostazioneDeposito].SupportPianoFerro.HMAX;
								WorkAreaState[NumPostazioneDeposito].Supporto.Tipologia 				:= CASSA_STANDARD;//ActualPickingListFromHMI.Support.Tipologia;
								WorkAreaState[NumPostazioneDeposito].Supporto.XDim 						:= RequestPickingListFromHMIWorkArea[NumPostazioneDeposito].SupportPianoFerro.XDim;
								WorkAreaState[NumPostazioneDeposito].Supporto.YDim 						:= RequestPickingListFromHMIWorkArea[NumPostazioneDeposito].SupportPianoFerro.YDim;
								WorkAreaState[NumPostazioneDeposito].Supporto.ZDim 						:= RequestPickingListFromHMIWorkArea[NumPostazioneDeposito].SupportPianoFerro.ZDim;
								WorkAreaOffset[NumPostazioneDeposito].Y 								:= OFFSET_POSTAZIONE_TELAIO - WorkAreaState[NumPostazioneDeposito].Supporto.YDim /2;//ATTENZIONE!!! per poter lavorare in centro con i supporti pari, questa misura è la distanza tra il riscontro bundle verticale e il centro postazione PARI
								
								WorkAreaProductionList[NumPostazioneDeposito].Support := WorkAreaState[NumPostazioneDeposito].Supporto;
							
								
								FOR j:= Iforstart TO Iforend DO
									IF NOT HMI_WorkAreaDataPicking[j].Destinazione THEN
										IF HMI_WorkAreaDataPicking[j].NumElementiDaLavorare >= 1 THEN
											
											ElementiDaDepositare[IdxLista] := ElementiElaborati[IdxLista] + HMI_WorkAreaDataPicking[j].NumElementiDaLavorare;
											FOR k := ElementiElaborati[IdxLista] TO ElementiDaDepositare[IdxLista]-1 DO	
												WorkAreaProductionList[NumPostazioneDeposito].PElementList[k].WA_PRELIEVO := j;
												WorkAreaProductionList[NumPostazioneDeposito].PElementList[k].WA_DEPOSITO := i;	
												ElementiElaborati[IdxLista] := ElementiElaborati[IdxLista]+1; 
											
												//Numero_Piezas_estacionPikin := 	Numero_Piezas_estacionPikin + ElementiDaDepositare[IdxLista] ;  
											END_FOR
												pr1 := 	Numero_Piezas_estacionPikin ;  
												pr2 := Numero_Piezas_estacionPikin  + HMI_WorkAreaDataPicking[j].NumElementiDaLavorare -1 ;				
											FOR ja := Numero_Piezas_estacionPikin  TO Numero_Piezas_estacionPikin  + HMI_WorkAreaDataPicking[j].NumElementiDaLavorare-1 DO
												// Se van Añadiendo los Diferentes Espesores de la receta del piking ######################################
												HMi_DimensionesPiezasWorkAreaDeposito[ja].Dim_Horizontal := RequestPickingListFromHMIWorkArea[j].SlabDimension ;
												//########################################################################################################		  
											END_FOR		  
												Numero_Piezas_estacionPikin := Numero_Piezas_estacionPikin +HMI_WorkAreaDataPicking[j].NumElementiDaLavorare; 			
											CASE HMI_WorkAreaDataPicking[j].Typology OF 
												(* Se ho una cassa pianale in legno *)
												LEGNO_PIANO:
													WorkAreaState[j].Supporto.Code 					:= ActualPickingListFromHMI[IdxLista].SupportPianoLegno.Code;
													WorkAreaState[j].Supporto.DimBaseUtile		 	:= RequestPickingListFromHMIWorkArea[j].SupportPianoLegno.DimBaseUtile;
													WorkAreaState[j].Supporto.AltezzaDenteRitenuta 	:= RequestPickingListFromHMIWorkArea[j].SupportPianoLegno.ZDim+20;
													WorkAreaState[j].Supporto.DimVertice 			:= RequestPickingListFromHMIWorkArea[j].SupportPianoLegno.DimVertice;
													WorkAreaState[j].Supporto.HMAX 					:= RequestPickingListFromHMIWorkArea[j].SupportPianoLegno.HMAX;
													WorkAreaState[j].Supporto.Tipologia 			:=  e_Tipo_Pallet.CASSA_STANDARD;//ActualPickingListFromHMI[1].Support.Tipologia;
													WorkAreaState[j].Supporto.XDim 					:= RequestPickingListFromHMIWorkArea[j].SupportPianoLegno.XDim;
													WorkAreaState[j].Supporto.YDim 					:= RequestPickingListFromHMIWorkArea[j].SupportPianoLegno.YDim;
													WorkAreaState[j].Supporto.ZDim 					:= RequestPickingListFromHMIWorkArea[j].SupportPianoLegno.ZDim;
													WorkAreaOffset[j].Y 							:= OFFSET_POSTAZIONE_LEGNO + WorkAreaState[j].Supporto.YDim/2;//ATTENZIONE!!! per poter lavorare in centro con i supporti pari, questa misura è la distanza tra il riscontro bundle verticale e il centro postazione PARI
												(* Se ho una cassa pianale in ferro su supporto *)
												TELAIO_PIANO:
													WorkAreaState[j].Supporto.Code 					:= ActualPickingListFromHMI[IdxLista].SupportPianoFerro.Code;
													WorkAreaState[j].Supporto.DimBaseUtile		 	:= RequestPickingListFromHMIWorkArea[j].SupportPianoFerro.DimBaseUtile;
													WorkAreaState[j].Supporto.AltezzaDenteRitenuta 	:= RequestPickingListFromHMIWorkArea[j].SupportPianoFerro.ZDim+20;
													WorkAreaState[j].Supporto.DimVertice 			:= RequestPickingListFromHMIWorkArea[j].SupportPianoFerro.DimVertice;
													WorkAreaState[j].Supporto.HMAX 					:= RequestPickingListFromHMIWorkArea[j].SupportPianoFerro.HMAX;
													WorkAreaState[j].Supporto.Tipologia 			:=  e_Tipo_Pallet.CASSA_STANDARD;//ActualPickingListFromHMI[1].Support.Tipologia;
													WorkAreaState[j].Supporto.XDim 					:= RequestPickingListFromHMIWorkArea[j].SupportPianoFerro.XDim;
													WorkAreaState[j].Supporto.YDim 					:= RequestPickingListFromHMIWorkArea[j].SupportPianoFerro.YDim;
													WorkAreaState[j].Supporto.ZDim 					:= RequestPickingListFromHMIWorkArea[j].SupportPianoFerro.ZDim;
													WorkAreaOffset[j].Y 							:= OFFSET_POSTAZIONE_TELAIO - WorkAreaState[j].Supporto.YDim/2;//ATTENZIONE!!! per poter lavorare in centro con i supporti pari, questa misura è la distanza tra il riscontro bundle verticale e il centro postazione PARI
												(* Se ho un bundle *)
												BUNDLE_VERT:
													//WorkAreaState[j].P := ElementiDaDepositare;
													WorkAreaState[j].Supporto.Code 					:= RequestPickingListFromHMIWorkArea[j].SupportVertBundle.Code;
													WorkAreaState[j].Supporto.DimBaseUtile		 	:= RequestPickingListFromHMIWorkArea[j].SupportVertBundle.DimBaseUtile;
													WorkAreaState[j].Supporto.AltezzaDenteRitenuta 	:= RequestPickingListFromHMIWorkArea[j].SupportVertBundle.ZDim+20;
													WorkAreaState[j].Supporto.DimVertice 			:= RequestPickingListFromHMIWorkArea[j].SupportVertBundle.DimVertice;
													WorkAreaState[j].Supporto.HMAX 					:= RequestPickingListFromHMIWorkArea[j].SupportVertBundle.HMAX;
													WorkAreaState[j].Supporto.Tipologia 			:= e_Tipo_Pallet.BUNDLE;//ActualPickingListFromHMI.SupportVertBundle.Tipologia;
													WorkAreaState[j].Supporto.XDim 					:= RequestPickingListFromHMIWorkArea[j].SupportVertBundle.XDim;
													WorkAreaState[j].Supporto.YDim 					:= RequestPickingListFromHMIWorkArea[j].SupportVertBundle.YDim;
													WorkAreaState[j].Supporto.ZDim 					:= RequestPickingListFromHMIWorkArea[j].SupportVertBundle.ZDim;
													WorkAreaState[j].Supporto.ZDim_Ext1        		:= WorkAreaState[j].Supporto.ZDim + 20;
													WorkAreaState[j].Supporto.TipoPianoAppoggio 	:= 1;                      
													WorkAreaState[j].Supporto.AltezzaDenteRitenuta	:= 20; 
													WorkAreaState[j].Supporto.LatoDeposito 			:= 180;   	
													  
													WorkAreaOffset[j].Y 							:= 0 ;	
												  
												A_FRAME_VERT:  						
													//WorkAreaState[j].P := ElementiDaDepositare;
													WorkAreaState[j].Supporto.Code 					:= ActualPickingListFromHMI[IdxLista].SupportVertCav.Code;
													WorkAreaState[j].Supporto.DimBaseUtile		 	:= RequestPickingListFromHMIWorkArea[j].SupportVertCav.DimBaseUtile;
													WorkAreaState[j].Supporto.AltezzaDenteRitenuta 	:= RequestPickingListFromHMIWorkArea[j].SupportVertCav.ZDim+20;
													WorkAreaState[j].Supporto.DimVertice 			:= RequestPickingListFromHMIWorkArea[j].SupportVertCav.DimVertice;
													WorkAreaState[j].Supporto.HMAX 					:= RequestPickingListFromHMIWorkArea[j].SupportVertcav.HMAX;
													WorkAreaState[j].Supporto.Tipologia 			:= CAVALLETTO;//ActualPickingListFromHMI.SupportVert.Tipologia;
													WorkAreaState[j].Supporto.XDim 					:= RequestPickingListFromHMIWorkArea[j].SupportVertCav.XDim;
													WorkAreaState[j].Supporto.YDim 					:= RequestPickingListFromHMIWorkArea[j].SupportVertCav.YDim;
													WorkAreaState[j].Supporto.ZDim 					:= RequestPickingListFromHMIWorkArea[j].SupportVertCav.ZDim;
													WorkAreaState[j].Supporto.ZDim_Ext1        		:= WorkAreaState[j].Supporto.ZDim + 20;	
													WorkAreaState[j].Supporto.TipoPianoAppoggio 	:= 1;                      
													WorkAreaState[j].Supporto.AltezzaDenteRitenuta	:= 15; 	
													WorkAreaState[j].Supporto.TipoTrabajoLado_Cavallete := HMI_WorkAreaDataPicking[j].TipoTrabajoLado_Cavallete ; 
													WorkAreaOffset[j].Y 							:= OFFSET_POSTAZIONE_LEGNO + WorkAreaState[j].Supporto.YDim/2;//ATTENZIONE!!! per poter lavorare in centro con i supporti pari, questa misura è la distanza tra il riscontro bundle verticale e il centro postazione PARI
											   		CoordenadaPasillo0_Y 							:= WorkArea[j].Y +  WorkAreaOffset[j].Y  - Dimensioni_Pinza.Spessore - INGOMBRO_RISCONTRO_FRAME - WorkAreaState[j].Supporto.YDim /2 ;
													CoordenadaPasillo180_Y 							:= WorkArea[j].Y + WorkAreaState[j].Supporto.YDim /2 + WorkAreaOffset[j].Y  + Dimensioni_Pinza.Spessore + INGOMBRO_RISCONTRO_FRAME  ;	
											END_CASE	
											WorkAreaProductionList[j].Support := WorkAreaState[j].Supporto; 
										END_IF
									END_IF     
									TFClearApprendimento(ADR(WorkAreaState[j].Apprendimento));//Azzeramento apprendimento 
								END_FOR
								EXIT; 
							(* Se ho un bundle *)
							BUNDLE_VERT:
								
								//Se ho deposito verticale su bundle
								
								WorkAreaState[NumPostazioneDeposito].Supporto.Code 						:= ActualPickingListFromHMI[IdxLista].SupportVertBundle.Code;
								WorkAreaState[NumPostazioneDeposito].Supporto.DimBaseUtile		 		:= RequestPickingListFromHMIWorkArea[NumPostazioneDeposito].SupportVertBundle.DimBaseUtile;
								WorkAreaState[NumPostazioneDeposito].Supporto.DimVertice 				:= RequestPickingListFromHMIWorkArea[NumPostazioneDeposito].SupportVertBundle.DimVertice;
								WorkAreaState[NumPostazioneDeposito].Supporto.HMAX 						:= RequestPickingListFromHMIWorkArea[NumPostazioneDeposito].SupportVertBundle.HMAX;
								WorkAreaState[NumPostazioneDeposito].Supporto.Tipologia 				:= e_Tipo_Pallet.BUNDLE;
								WorkAreaState[NumPostazioneDeposito].Supporto.XDim 						:= RequestPickingListFromHMIWorkArea[NumPostazioneDeposito].SupportVertBundle.XDim;
								WorkAreaState[NumPostazioneDeposito].Supporto.YDim 						:= RequestPickingListFromHMIWorkArea[NumPostazioneDeposito].SupportVertBundle.YDim;
								WorkAreaState[NumPostazioneDeposito].Supporto.ZDim 						:= RequestPickingListFromHMIWorkArea[NumPostazioneDeposito].SupportVertBundle.ZDim;
								WorkAreaState[NumPostazioneDeposito].Supporto.TipoPianoAppoggio 		:= 1;                      
								WorkAreaState[NumPostazioneDeposito].Supporto.AltezzaDenteRitenuta		:= 20; 
								WorkAreaState[NumPostazioneDeposito].Supporto.LatoDeposito 				:= 180; 
											   
								WorkAreaProductionList[NumPostazioneDeposito].Support 					:= WorkAreaState[NumPostazioneDeposito].Supporto;
								
								FOR j:= Iforstart TO Iforend DO
									IF NOT HMI_WorkAreaDataPicking[j].Destinazione THEN
										IF HMI_WorkAreaDataPicking[j].NumElementiDaLavorare >= 1 THEN
												 
											ElementiDaDepositare[IdxLista] := ElementiElaborati[IdxLista] + HMI_WorkAreaDataPicking[j].NumElementiDaLavorare;
											FOR k := ElementiElaborati[IdxLista] TO ElementiDaDepositare[IdxLista]-1 DO	
												WorkAreaProductionList[NumPostazioneDeposito].PElementList[k].WA_PRELIEVO := j;
												WorkAreaProductionList[NumPostazioneDeposito].PElementList[k].WA_DEPOSITO := i;	
												ElementiElaborati[IdxLista] := ElementiElaborati[IdxLista]+1; 
											END_FOR
												pr1 := 	Numero_Piezas_estacionPikin ;  
												pr2 := Numero_Piezas_estacionPikin  + HMI_WorkAreaDataPicking[j].NumElementiDaLavorare -1 ;				
											FOR ja := Numero_Piezas_estacionPikin  TO Numero_Piezas_estacionPikin  + HMI_WorkAreaDataPicking[j].NumElementiDaLavorare-1 DO
												// Se van Añadiendo los Diferentes Espesores de la receta del piking ######################################
												HMi_DimensionesPiezasWorkAreaDeposito[ja].Dim_Horizontal := RequestPickingListFromHMIWorkArea[j].SlabDimension ;
												//########################################################################################################		  
											END_FOR		  
												Numero_Piezas_estacionPikin := Numero_Piezas_estacionPikin +HMI_WorkAreaDataPicking[j].NumElementiDaLavorare; 	 
											CASE HMI_WorkAreaDataPicking[j].Typology OF 
												(* Se ho una cassa pianale in legno *)
												LEGNO_PIANO:
													WorkAreaState[j].Supporto.Code 					:= ActualPickingListFromHMI[IdxLista].SupportPianoLegno.Code;
													WorkAreaState[j].Supporto.DimBaseUtile		 	:= RequestPickingListFromHMIWorkArea[j].SupportPianoLegno.DimBaseUtile;
													WorkAreaState[j].Supporto.AltezzaDenteRitenuta 	:= RequestPickingListFromHMIWorkArea[j].SupportPianoLegno.ZDim+20;
													WorkAreaState[j].Supporto.DimVertice 			:= RequestPickingListFromHMIWorkArea[j].SupportPianoLegno.DimVertice;
													WorkAreaState[j].Supporto.HMAX 					:= RequestPickingListFromHMIWorkArea[j].SupportPianoLegno.HMAX;
													WorkAreaState[j].Supporto.Tipologia 			:=  e_Tipo_Pallet.CASSA_STANDARD;//ActualPickingListFromHMI[1].Support.Tipologia;
													WorkAreaState[j].Supporto.XDim 					:= RequestPickingListFromHMIWorkArea[j].SupportPianoLegno.XDim;
													WorkAreaState[j].Supporto.YDim 					:= RequestPickingListFromHMIWorkArea[j].SupportPianoLegno.YDim;
													WorkAreaState[j].Supporto.ZDim 					:= RequestPickingListFromHMIWorkArea[j].SupportPianoLegno.ZDim;
													WorkAreaOffset[j].Y 							:= OFFSET_POSTAZIONE_LEGNO + WorkAreaState[j].Supporto.YDim/2;//ATTENZIONE!!! per poter lavorare in centro con i supporti pari, questa misura è la distanza tra il riscontro bundle verticale e il centro postazione PARI
												(* Se ho una cassa pianale in ferro su supporto *)
												TELAIO_PIANO:
													WorkAreaState[j].Supporto.Code 					:= ActualPickingListFromHMI[IdxLista].SupportPianoFerro.Code;
													WorkAreaState[j].Supporto.DimBaseUtile		 	:= RequestPickingListFromHMIWorkArea[j].SupportPianoFerro.DimBaseUtile;
													WorkAreaState[j].Supporto.AltezzaDenteRitenuta 	:= RequestPickingListFromHMIWorkArea[j].SupportPianoFerro.ZDim+20;
													WorkAreaState[j].Supporto.DimVertice 			:= RequestPickingListFromHMIWorkArea[j].SupportPianoFerro.DimVertice;
													WorkAreaState[j].Supporto.HMAX 					:= RequestPickingListFromHMIWorkArea[j].SupportPianoFerro.HMAX;
													WorkAreaState[j].Supporto.Tipologia 			:=  e_Tipo_Pallet.CASSA_STANDARD;//ActualPickingListFromHMI[1].Support.Tipologia;
													WorkAreaState[j].Supporto.XDim 					:= RequestPickingListFromHMIWorkArea[j].SupportPianoFerro.XDim;
													WorkAreaState[j].Supporto.YDim 					:= RequestPickingListFromHMIWorkArea[j].SupportPianoFerro.YDim;
													WorkAreaState[j].Supporto.ZDim 					:= RequestPickingListFromHMIWorkArea[j].SupportPianoFerro.ZDim;
													WorkAreaOffset[j].Y 							:= OFFSET_POSTAZIONE_TELAIO - WorkAreaState[j].Supporto.YDim/2;//ATTENZIONE!!! per poter lavorare in centro con i supporti pari, questa misura è la distanza tra il riscontro bundle verticale e il centro postazione PARI
												(* Se ho un bundle *)
												BUNDLE_VERT:
													//WorkAreaState[j].P := ElementiDaDepositare;
													WorkAreaState[j].Supporto.Code 					:= ActualPickingListFromHMI[IdxLista].SupportVertBundle.Code;
													WorkAreaState[j].Supporto.DimBaseUtile		 	:= RequestPickingListFromHMIWorkArea[j].SupportVertBundle.DimBaseUtile;
													WorkAreaState[j].Supporto.AltezzaDenteRitenuta 	:= RequestPickingListFromHMIWorkArea[j].SupportVertBundle.ZDim+20;
													WorkAreaState[j].Supporto.DimVertice 			:= RequestPickingListFromHMIWorkArea[j].SupportVertBundle.DimVertice;
													WorkAreaState[j].Supporto.HMAX 					:= RequestPickingListFromHMIWorkArea[j].SupportVertBundle.HMAX;
													WorkAreaState[j].Supporto.Tipologia 			:= e_Tipo_Pallet.BUNDLE;//ActualPickingListFromHMI.SupportVert.Tipologia;
													WorkAreaState[j].Supporto.XDim 					:= RequestPickingListFromHMIWorkArea[j].SupportVertBundle.XDim;
													WorkAreaState[j].Supporto.YDim 					:= RequestPickingListFromHMIWorkArea[j].SupportVertBundle.YDim;
													WorkAreaState[j].Supporto.ZDim 					:= RequestPickingListFromHMIWorkArea[j].SupportVertBundle.ZDim;
													WorkAreaState[j].Supporto.ZDim_Ext1        		:= WorkAreaState[j].Supporto.ZDim + 20;	
													// **Lo Que Habia	
													WorkAreaOffset[j].Y 							:= 0;
													//Mod 25/&/2025	  
													//WorkAreaOffset[j].Y 		:= ActualPickingListFromHMI[IdxLista].SupportVertBundle.YDim-ActualPickingListFromHMI[IdxLista].SupportVertBundle.DimBaseUtile -40;	
			
												(* Se ho un A_Frame *)	  
												A_FRAME_VERT:  						
													//WorkAreaState[j].P := ElementiDaDepositare;
													WorkAreaState[j].Supporto.Code 					:= ActualPickingListFromHMI[IdxLista].SupportVertCav.Code;
													WorkAreaState[j].Supporto.DimBaseUtile		 	:= RequestPickingListFromHMIWorkArea[j].SupportVertCav.DimBaseUtile;
													WorkAreaState[j].Supporto.AltezzaDenteRitenuta 	:= RequestPickingListFromHMIWorkArea[j].SupportVertCav.ZDim+20;
													WorkAreaState[j].Supporto.DimVertice 			:= RequestPickingListFromHMIWorkArea[j].SupportVertCav.DimVertice;
													WorkAreaState[j].Supporto.HMAX 					:= RequestPickingListFromHMIWorkArea[j].SupportVertCav.HMAX;
													WorkAreaState[j].Supporto.Tipologia 			:= CAVALLETTO;//ActualPickingListFromHMI.SupportVert.Tipologia;
													WorkAreaState[j].Supporto.XDim 					:= RequestPickingListFromHMIWorkArea[j].SupportVertCav.XDim;
													WorkAreaState[j].Supporto.YDim 					:= RequestPickingListFromHMIWorkArea[j].SupportVertCav.YDim;
													WorkAreaState[j].Supporto.ZDim 					:= RequestPickingListFromHMIWorkArea[j].SupportVertCav.ZDim;
													WorkAreaState[j].Supporto.ZDim_Ext1        		:= WorkAreaState[j].Supporto.ZDim + 20;	
													WorkAreaState[j].Supporto.TipoPianoAppoggio 	:= 1;                      
													WorkAreaState[j].Supporto.AltezzaDenteRitenuta	:= 15; 	
													WorkAreaState[j].Supporto.TipoTrabajoLado_Cavallete := HMI_WorkAreaDataPicking[j].TipoTrabajoLado_Cavallete ; 
													WorkAreaOffset[j].Y 							:= OFFSET_POSTAZIONE_LEGNO + WorkAreaState[j].Supporto.YDim/2;//ATTENZIONE!!! per poter lavorare in centro con i supporti pari, questa misura è la distanza tra il riscontro bundle verticale e il centro postazione PARI
													CoordenadaPasillo0_Y 							:= WorkArea[j].Y +  WorkAreaOffset[j].Y  - Dimensioni_Pinza.Spessore - INGOMBRO_RISCONTRO_FRAME - WorkAreaState[j].Supporto.YDim /2 ;
													CoordenadaPasillo180_Y 							:= WorkArea[j].Y + WorkAreaState[j].Supporto.YDim /2 + WorkAreaOffset[j].Y  + Dimensioni_Pinza.Spessore + INGOMBRO_RISCONTRO_FRAME  ;		  
											END_CASE
											//WorkAreaProductionList[j].Support := HMI_Formatura.HMI_Forming_Supporto;		  
											WorkAreaProductionList[j].Support := WorkAreaState[j].Supporto;
										END_IF
									END_IF
									TFClearApprendimento(ADR(WorkAreaState[j].Apprendimento));//Azzeramento apprendimento
								END_FOR
								EXIT; 
							(* Se ho un A_Frame *)	
							A_FRAME_VERT:
								
								WorkAreaState[NumPostazioneDeposito].Supporto.Code 						:= ActualPickingListFromHMI[IdxLista].SupportVertCav.Code;
								WorkAreaState[NumPostazioneDeposito].Supporto.DimBaseUtile		 		:= RequestPickingListFromHMIWorkArea[NumPostazioneDeposito].SupportVertCav.DimBaseUtile;
								WorkAreaState[NumPostazioneDeposito].Supporto.DimVertice 				:= RequestPickingListFromHMIWorkArea[NumPostazioneDeposito].SupportVertCav.DimVertice;
								WorkAreaState[NumPostazioneDeposito].Supporto.HMAX 						:= RequestPickingListFromHMIWorkArea[NumPostazioneDeposito].SupportVertCav.HMAX;
								WorkAreaState[NumPostazioneDeposito].Supporto.Tipologia 				:= e_Tipo_Pallet.CAVALLETTO;//ActualPickingListFromHMI.SupportVertBundle.Tipologia;
								WorkAreaState[NumPostazioneDeposito].Supporto.XDim 						:= RequestPickingListFromHMIWorkArea[NumPostazioneDeposito].SupportVertCav.XDim;
								WorkAreaState[NumPostazioneDeposito].Supporto.YDim 						:= RequestPickingListFromHMIWorkArea[NumPostazioneDeposito].SupportVertCav.YDim;
								WorkAreaState[NumPostazioneDeposito].Supporto.ZDim 						:= RequestPickingListFromHMIWorkArea[NumPostazioneDeposito].SupportVertCav.ZDim;
								WorkAreaState[NumPostazioneDeposito].Supporto.TipoPianoAppoggio 		:= 1;                      
								WorkAreaState[NumPostazioneDeposito].Supporto.AltezzaDenteRitenuta		:= 15; 
								WorkAreaState[NumPostazioneDeposito].Supporto.TipoTrabajoLado_Cavallete 					:= HMI_WorkAreaDataPicking[NumPostazioneDeposito].TipoTrabajoLado_Cavallete ; 
								//WorkAreaOffset[NumPostazioneDeposito].Y 								:= OFFSET_POSTAZIONE_LEGNO (*- ActualPickingListFromHMI[IdxLista].SupportPianoFerro.YDim/2*);
								WorkAreaOffset[NumPostazioneDeposito].Y 								:= OFFSET_POSTAZIONE_LEGNO + WorkAreaState[NumPostazioneDeposito].Supporto.YDim/2;	
								CoordenadaPasillo0_Y := WorkArea[NumPostazioneDeposito].Y +  WorkAreaOffset[NumPostazioneDeposito].Y  - Dimensioni_Pinza.Spessore - INGOMBRO_RISCONTRO_BUNDLE - WorkAreaState[NumPostazioneDeposito].Supporto.YDim /2 ;
								CoordenadaPasillo180_Y := WorkArea[NumPostazioneDeposito].Y + WorkAreaState[NumPostazioneDeposito].Supporto.YDim /2 + WorkAreaOffset[NumPostazioneDeposito].Y  + Dimensioni_Pinza.Spessore + INGOMBRO_RISCONTRO_FRAME  ;	
								WorkAreaProductionList[NumPostazioneDeposito].Support 				:= WorkAreaState[NumPostazioneDeposito].Supporto; 
								
								FOR j:= Iforstart TO Iforend DO
									IF NOT HMI_WorkAreaDataPicking[j].Destinazione THEN
										IF HMI_WorkAreaDataPicking[j].NumElementiDaLavorare >= 1 THEN
										ElementiDaDepositare[IdxLista] := ElementiElaborati[IdxLista] + HMI_WorkAreaDataPicking[j].NumElementiDaLavorare;
											FOR k := ElementiElaborati[IdxLista] TO ElementiDaDepositare[IdxLista]-1 DO	
												WorkAreaProductionList[NumPostazioneDeposito].PElementList[k].WA_PRELIEVO := j;
												WorkAreaProductionList[NumPostazioneDeposito].PElementList[k].WA_DEPOSITO := i;	
												ElementiElaborati[IdxLista] := ElementiElaborati[IdxLista]+1; 
											END_FOR 
													  
																
												CASE HMI_WorkAreaDataPicking[NumPostazioneDeposito].TipoTrabajoLado_Cavallete OF
												0:
													pr1 := Numero_piezas_CaballeteEstacionPiking.HMI_NumeroPezziPresentiPostazione_A_Cavaleto ; 
													pr2 := Numero_piezas_CaballeteEstacionPiking.HMI_NumeroPezziPresentiPostazione_B_Cavaleto ;  
													FOR ja := Numero_piezas_CaballeteEstacionPiking.HMI_NumeroPezziPresentiPostazione_A_Cavaleto  TO Numero_piezas_CaballeteEstacionPiking.HMI_NumeroPezziPresentiPostazione_A_Cavaleto  + HMI_WorkAreaDataPicking[j].NumElementiDaLavorare-1 DO
														  Fun_PiezaLadoCaballete(Nu_PiezaGlobal:= ja , Nu_pieza_LadoA=> P_ladoA , Nu_pieza_LadoB=> P_ladoB , Grados := ADR(LadoRegistar));
														IF  LadoRegistar  = 0 THEN 
															
															HMi_DimensionesPiezasWorkAreaDeposito[P_ladoA].DimPieza_LadoA := RequestPickingListFromHMIWorkArea[j].SlabDimension ;
														ELSIF LadoRegistar  = 180 THEN 	
															HMi_DimensionesPiezasWorkAreaDeposito[P_ladoB].DimPieza_LadoB := RequestPickingListFromHMIWorkArea[j].SlabDimension ;		  
														END_IF
													END_FOR		  
													Numero_piezas_CaballeteEstacionPiking.HMI_NumeroPezziPresentiPostazione_A_Cavaleto := Numero_piezas_CaballeteEstacionPiking.HMI_NumeroPezziPresentiPostazione_A_Cavaleto + HMI_WorkAreaDataPicking[j].NumElementiDaLavorare; 	
												1:
													FOR ja := Numero_piezas_CaballeteEstacionPiking.HMI_NumeroPezziPresentiPostazione_A_Cavaleto  TO Numero_piezas_CaballeteEstacionPiking.HMI_NumeroPezziPresentiPostazione_A_Cavaleto  + HMI_WorkAreaDataPicking[j].NumElementiDaLavorare-1 DO
														// Se van Añadiendo los Diferentes Espesores de la receta del piking ######################################
														HMi_DimensionesPiezasWorkAreaDeposito[ja].DimPieza_LadoA := RequestPickingListFromHMIWorkArea[j].SlabDimension ;
														//########################################################################################################	
													END_FOR		  
													Numero_piezas_CaballeteEstacionPiking.HMI_NumeroPezziPresentiPostazione_A_Cavaleto := Numero_piezas_CaballeteEstacionPiking.HMI_NumeroPezziPresentiPostazione_A_Cavaleto + HMI_WorkAreaDataPicking[j].NumElementiDaLavorare; 		  	  	  
													;
												2:
													FOR ja := Numero_piezas_CaballeteEstacionPiking.HMI_NumeroPezziPresentiPostazione_B_Cavaleto  TO Numero_piezas_CaballeteEstacionPiking.HMI_NumeroPezziPresentiPostazione_B_Cavaleto  + HMI_WorkAreaDataPicking[j].NumElementiDaLavorare-1 DO
														// Se van Añadiendo los Diferentes Espesores de la receta del piking ######################################
														HMi_DimensionesPiezasWorkAreaDeposito[ja].DimPieza_LadoB := RequestPickingListFromHMIWorkArea[j].SlabDimension ;
														//########################################################################################################	
													END_FOR		  
													Numero_piezas_CaballeteEstacionPiking.HMI_NumeroPezziPresentiPostazione_B_Cavaleto := Numero_piezas_CaballeteEstacionPiking.HMI_NumeroPezziPresentiPostazione_B_Cavaleto + HMI_WorkAreaDataPicking[j].NumElementiDaLavorare; 			  	  	
													;		  
											END_CASE
											
															  
																
																		  
									
											CASE HMI_WorkAreaDataPicking[j].Typology OF 
												(* Se ho una cassa pianale in legno *)
												LEGNO_PIANO:
													WorkAreaState[j].Supporto.Code 					:= ActualPickingListFromHMI[IdxLista].SupportPianoLegno.Code;
													WorkAreaState[j].Supporto.DimBaseUtile		 	:= RequestPickingListFromHMIWorkArea[j].SupportPianoLegno.DimBaseUtile;
													WorkAreaState[j].Supporto.AltezzaDenteRitenuta 	:= RequestPickingListFromHMIWorkArea[j].SupportPianoLegno.ZDim+20;
													WorkAreaState[j].Supporto.DimVertice 			:= RequestPickingListFromHMIWorkArea[j].SupportPianoLegno.DimVertice;
													WorkAreaState[j].Supporto.HMAX 					:= RequestPickingListFromHMIWorkArea[j].SupportPianoLegno.HMAX;
													WorkAreaState[j].Supporto.Tipologia 			:=  e_Tipo_Pallet.CASSA_STANDARD;//ActualPickingListFromHMI[1].Support.Tipologia;
													WorkAreaState[j].Supporto.XDim 					:= RequestPickingListFromHMIWorkArea[j].SupportPianoLegno.XDim;
													WorkAreaState[j].Supporto.YDim 					:= RequestPickingListFromHMIWorkArea[j].SupportPianoLegno.YDim;
													WorkAreaState[j].Supporto.ZDim 					:= RequestPickingListFromHMIWorkArea[j].SupportPianoLegno.ZDim;
													WorkAreaOffset[j].Y 							:= OFFSET_POSTAZIONE_LEGNO + WorkAreaState[j].Supporto.YDim/2;//ATTENZIONE!!! per poter lavorare in centro con i supporti pari, questa misura è la distanza tra il riscontro bundle verticale e il centro postazione PARI
												(* Se ho una cassa pianale in ferro su supporto *)
												TELAIO_PIANO:
													WorkAreaState[j].Supporto.Code 					:= ActualPickingListFromHMI[IdxLista].SupportPianoFerro.Code;
													WorkAreaState[j].Supporto.DimBaseUtile		 	:= RequestPickingListFromHMIWorkArea[j].SupportPianoFerro.DimBaseUtile;
													WorkAreaState[j].Supporto.AltezzaDenteRitenuta 	:= RequestPickingListFromHMIWorkArea[j].SupportPianoFerro.ZDim+20;
													WorkAreaState[j].Supporto.DimVertice 			:= RequestPickingListFromHMIWorkArea[j].SupportPianoFerro.DimVertice;
													WorkAreaState[j].Supporto.HMAX 					:= RequestPickingListFromHMIWorkArea[j].SupportPianoFerro.HMAX;
													WorkAreaState[j].Supporto.Tipologia 			:=  e_Tipo_Pallet.CASSA_STANDARD;//ActualPickingListFromHMI[1].Support.Tipologia;
													WorkAreaState[j].Supporto.XDim 					:= RequestPickingListFromHMIWorkArea[j].SupportPianoFerro.XDim;
													WorkAreaState[j].Supporto.YDim 					:= RequestPickingListFromHMIWorkArea[j].SupportPianoFerro.YDim;
													WorkAreaState[j].Supporto.ZDim 					:= RequestPickingListFromHMIWorkArea[j].SupportPianoFerro.ZDim;
													WorkAreaOffset[j].Y 							:= OFFSET_POSTAZIONE_TELAIO - WorkAreaState[j].Supporto.YDim/2;//ATTENZIONE!!! per poter lavorare in centro con i supporti pari, questa misura è la distanza tra il riscontro bundle verticale e il centro postazione PARI
												(* Se ho un bundle *)
												BUNDLE_VERT:
													//WorkAreaState[j].P := ElementiDaDepositare;
													WorkAreaState[j].Supporto.Code 					:= ActualPickingListFromHMI[IdxLista].SupportVertBundle.Code;
													WorkAreaState[j].Supporto.DimBaseUtile		 	:= RequestPickingListFromHMIWorkArea[j].SupportVertBundle.DimBaseUtile;
													WorkAreaState[j].Supporto.AltezzaDenteRitenuta 	:= RequestPickingListFromHMIWorkArea[j].SupportVertBundle.ZDim+20;
													WorkAreaState[j].Supporto.DimVertice 			:= RequestPickingListFromHMIWorkArea[j].SupportVertBundle.DimVertice;
													WorkAreaState[j].Supporto.HMAX 					:= RequestPickingListFromHMIWorkArea[j].SupportVertBundle.HMAX;
													WorkAreaState[j].Supporto.Tipologia 			:= e_Tipo_Pallet.BUNDLE;//ActualPickingListFromHMI.SupportVert.Tipologia;
													WorkAreaState[j].Supporto.XDim 					:= RequestPickingListFromHMIWorkArea[j].SupportVertBundle.XDim;
													WorkAreaState[j].Supporto.YDim 					:= RequestPickingListFromHMIWorkArea[j].SupportVertBundle.YDim;
													WorkAreaState[j].Supporto.ZDim 					:= RequestPickingListFromHMIWorkArea[j].SupportVertBundle.ZDim;
													WorkAreaState[j].Supporto.ZDim_Ext1        		:= WorkAreaState[j].Supporto.ZDim + 20;	
													WorkAreaState[j].Supporto.TipoPianoAppoggio 	:= 1;                      
													WorkAreaState[j].Supporto.AltezzaDenteRitenuta	:= 20; 
													WorkAreaState[j].Supporto.LatoDeposito 			:= 180; 
													//**Lo Que Habia
													WorkAreaOffset[j].Y 							:= 0;
													//Mod 25/&/2025	  
													//WorkAreaOffset[j].Y 		:= ActualPickingListFromHMI[IdxLista].SupportVertBundle.YDim-ActualPickingListFromHMI[IdxLista].SupportVertBundle.DimBaseUtile -40;					
												(* Se ho un A_Frame *)	  
												A_FRAME_VERT:  						
													//WorkAreaState[j].P := ElementiDaDepositare;
													WorkAreaState[j].Supporto.Code 					:= ActualPickingListFromHMI[IdxLista].SupportVertCav.Code;
													WorkAreaState[j].Supporto.DimBaseUtile		 	:= RequestPickingListFromHMIWorkArea[j].SupportVertCav.DimBaseUtile;
													WorkAreaState[j].Supporto.AltezzaDenteRitenuta 	:= RequestPickingListFromHMIWorkArea[j].SupportVertCav.ZDim+20;
													WorkAreaState[j].Supporto.DimVertice 			:= RequestPickingListFromHMIWorkArea[j].SupportVertCav.DimVertice;
													WorkAreaState[j].Supporto.HMAX 					:= RequestPickingListFromHMIWorkArea[j].SupportVertCav.HMAX;
													WorkAreaState[j].Supporto.Tipologia 			:= CAVALLETTO;//ActualPickingListFromHMI.SupportVertCav.Tipologia;
													WorkAreaState[j].Supporto.XDim 					:= RequestPickingListFromHMIWorkArea[j].SupportVertCav.XDim;
													WorkAreaState[j].Supporto.YDim 					:= RequestPickingListFromHMIWorkArea[j].SupportVertCav.YDim;
													WorkAreaState[j].Supporto.ZDim 					:= RequestPickingListFromHMIWorkArea[j].SupportVertCav.ZDim;
													WorkAreaState[j].Supporto.ZDim_Ext1        		:= WorkAreaState[j].Supporto.ZDim + 20;	
													WorkAreaState[j].Supporto.TipoPianoAppoggio 	:= 1;                      
													WorkAreaState[j].Supporto.AltezzaDenteRitenuta	:= 15; 	
													WorkAreaState[j].Supporto.TipoTrabajoLado_Cavallete := HMI_WorkAreaDataPicking[j].TipoTrabajoLado_Cavallete ; 	
													WorkAreaOffset[j].Y 							:= OFFSET_POSTAZIONE_LEGNO + WorkAreaState[j].Supporto.YDim /2;//ATTENZIONE!!! per poter lavorare in centro con i supporti pari, questa misura è la distanza tra il riscontro bundle verticale e il centro postazione PARI
												   	CoordenadaPasillo0_Y 							:= WorkArea[j].Y +  WorkAreaOffset[j].Y  - Dimensioni_Pinza.Spessore - INGOMBRO_RISCONTRO_FRAME - WorkAreaState[j].Supporto.YDim /2 ;
													CoordenadaPasillo180_Y 							:= WorkArea[j].Y + WorkAreaState[j].Supporto.YDim /2 + WorkAreaOffset[j].Y  + Dimensioni_Pinza.Spessore + INGOMBRO_RISCONTRO_FRAME  ;	
												
											END_CASE
													  
											WorkAreaProductionList[j].Support := WorkAreaState[j].Supporto;
										END_IF
									END_IF
									TFClearApprendimento(ADR(WorkAreaState[j].Apprendimento));//Azzeramento apprendimento
								END_FOR
								EXIT; 
						END_CASE // case Pricipal1
					END_IF	//-------->	 //-------> Palet destino
				END_FOR//----------For 1 HMI_WorkAreaDataPicking[i].Destinazione 
				
				Picking.Cmd_CalcolaLista[IdxLista] := TRUE;
				HMI_Forming_Attivazione[IdxLista] := TRUE;//attivo nuova formatura
			END_IF //------------------------------ActualPickingListFromHMI[IdxLista].State = e_StatoWorkOrder.DA_ESEGUIRE 
{endregion }
			 
{Region "Formaciones Nuevas" }
IF Picking.Cmd_CalcolaLista[IdxLista] AND HMI_Forming_Attivazione[IdxLista] AND NOT FormacionesCalculadas AND NOT FormacionPikingCalculada THEN
	idxForm:= IdxLista;		 
	CalFor := NumPostazioneDeposito;
{Region " calculo la formacion para los calculos "}
		  
	IF CalFor = NumPostazioneDeposito AND NOT FormacionPikingCalculada THEN // calcula la formacion para la estacion de piking
		MEMSET(destAddr := ADR(TFCalcoloFormaturaWA[CalFor]),fillByte := 0 , n := SIZEOF(TFCalcoloFormaturaWA[CalFor]));
		TFCalcoloFormaturaWA[CalFor].PulisciMemoria 			:= TRUE ; 
		TFCalcoloFormaturaWA[CalFor]();			   
		
			//Ponemos El tipo de soporte que tiene la estacion 
			HMI_Formatura.HMI_Forming_Supporto.Code				:= WorkAreaState[CalFor].Supporto.Code;
			HMI_Formatura.HMI_Forming_Supporto.XDim				:= WorkAreaState[CalFor].Supporto.XDim;
			HMI_Formatura.HMI_Forming_Supporto.YDim				:= WorkAreaState[CalFor].Supporto.YDim;
			HMI_Formatura.HMI_Forming_Supporto.ZDim				:= WorkAreaState[CalFor].Supporto.ZDim;
			HMI_Formatura.HMI_Forming_Supporto.DimBaseUtile		:= WorkAreaState[CalFor].Supporto.DimBaseUtile;
			HMI_Formatura.HMI_Forming_Supporto.DimVertice 		:= WorkAreaState[CalFor].Supporto.DimVertice;
			HMI_Formatura.HMI_Forming_Supporto.HMAX 			:= WorkAreaState[CalFor].Supporto.HMAX;
			HMI_Formatura.HMI_Forming_Supporto.Tipologia		:= WorkAreaState[CalFor].Supporto.Tipologia;// RequestPickingListFromHMI[1].Support.Tipologia;		
			CASE HMI_WorkAreaDataPicking[NumPostazioneDeposito].Typology OF 
				A_FRAME_VERT:
					HMI_Formatura.HMI_Forming_Supporto.TipoTrabajoLado_Cavallete :=	WorkAreaState[CalFor].Supporto.TipoTrabajoLado_Cavallete ;	   
					HMI_Formatura.HMI_Forming_Supporto.TipoPianoAppoggio 		:= 1;                      
					HMI_Formatura.HMI_Forming_Supporto.AltezzaDenteRitenuta		:= 15;              
					HMI_Formatura.HMI_Forming_Supporto.ZDim_Ext1        := HMI_Formatura.HMI_Forming_Supporto.ZDim + HMI_Formatura.HMI_Forming_Supporto.AltezzaDenteRitenuta;		  
				BUNDLE_VERT:
					HMI_Formatura.HMI_Forming_Supporto.YDim				:= WorkAreaState[CalFor].Supporto.YDim * 2;
					HMI_Formatura.HMI_Forming_Supporto.DimVertice 		:= WorkAreaState[CalFor].Supporto.DimVertice *2;	
					HMI_Formatura.HMI_Forming_Supporto.TipoPianoAppoggio := 1;                      
					HMI_Formatura.HMI_Forming_Supporto.AltezzaDenteRitenuta		:= 20;              
					HMI_Formatura.HMI_Forming_Supporto.ZDim_Ext1        := HMI_Formatura.HMI_Forming_Supporto.ZDim +	HMI_Formatura.HMI_Forming_Supporto.AltezzaDenteRitenuta;
			END_CASE
			//Copiamos es soporte en la lista de produccio Para le estacion de picking
			WorkAreaProductionList[CalFor].Support := HMI_Formatura.HMI_Forming_Supporto;
			//Añadimos las dikmensiones de la pieza	
			HMI_Formatura.HMI_Forming_LastraDaDepositare.XDim		:= RequestPickingListFromHMIWorkArea[CalFor].SlabDimension.XDim;
			HMI_Formatura.HMI_Forming_LastraDaDepositare.YDim		:= RequestPickingListFromHMIWorkArea[CalFor].SlabDimension.YDim;
			HMI_Formatura.HMI_Forming_LastraDaDepositare.ZDim		:= RequestPickingListFromHMIWorkArea[CalFor].SlabDimension.ZDim;
			//Escribimos el codigo para la estacion 
			HMI_Formatura.HMI_Forming_CodiciAbilitatiFormatura[IdxLista].Code[1] := 1; 
			// ########para quitar ###############################################################               
			FaldaDaDepositare.TypologyCode := RequestPickingListFromHMI[IdxLista].Layer.Tipologia;
			FaldaDaDepositare.XDim := RequestPickingListFromHMI[IdxLista].Layer.XDim;
			FaldaDaDepositare.YDim := RequestPickingListFromHMI[IdxLista].Layer.YDim;
			FaldaDaDepositare.ZDim := RequestPickingListFromHMI[IdxLista].Layer.ZDim;
			//#################################################################################
			//Vado ad assegnare il numero giusto di elementi a seconda se è presente o meno la falda 
			IF (RequestPickingListFromHMI[IdxLista].LayerSequence = 1 AND HMI_AbilitaDepositoFalda) AND RequestPickingListFromHMI[IdxLista].SupportPianoLegno.Tipologia <> CAVALLETTO AND RequestPickingListFromHMI[IdxLista].SupportPianoLegno.Tipologia <> BUNDLE THEN 
				HMI_Formatura.HMI_Forming_NumeroElementiDaDepositare	:= TO_UINT(2*RequestPickingListFromHMI[IdxLista].SlabNumber - 1);
			ELSE 
				HMI_Formatura.HMI_Forming_NumeroElementiDaDepositare	:= TO_UINT(RequestPickingListFromHMI[IdxLista].SlabNumber);
			END_IF
			//Ack 
				IF HMI_ErrAckCalcolaFormatura THEN
					HMI_Forming_ErroreCalcoli := 0;
					HMI_ErrAckCalcolaFormatura := FALSE;
					FOR i:= 1 TO MAXFORMING DO
						HMI_ConfermaAttivazioneFormatura[i] := FALSE;
						HMI_Forming_FormaturaAttivata[i] := FALSE;
					END_FOR
				END_IF
				
				//Azzeramento comandi in caso di errore
				IF HMI_Forming_ErroreCalcoli <> 0 THEN
					FOR i:=1 TO MAXFORMING DO
						HMI_Forming_Attivazione[i] 		:= FALSE;
						HMI_Forming_Disattivazione[i] 	:= FALSE;
					END_FOR
					HMI_Forming_Calcola 			:= FALSE;
				END_IF
				
			 
		END_IF 
{endregion}
			   
	IF  TFCalcoloFormaturaWA[CalFor].PulisciMemoria AND (TFCalcoloFormaturaWA[CalFor].PulisciMemoriaDone OR TRUE)AND NOT FormacionPikingCalculada THEN 
		HMI_Forming_FormaturaAttivata[CalFor] 	:= FALSE;	
		HMI_Forming_ErroreCalcoli := 0;	
		TFCalcoloFormaturaWA[CalFor].PulisciMemoria := FALSE ;
		IF (RequestPickingListFromHMI[1].LayerSequence = 0 OR NOT HMI_AbilitaDepositoFalda)
						AND HMI_Forming_NumeroElementiDaDepositare >0  THEN
			//Assegno l'ordine tutto a 1 perchè ho solo lastre	
			FOR i:= 1 TO MAXFORMINGSLAB DO
				//IF i <= HMI_Forming_NumeroElementiDaDepositare THEN
				IF i <= HMI_Forming_NumeroElementiDaDepositare + HMI_NumeroPezziPresentiPostazione[CalFor] THEN
				//IF i <= 20THEN
					TFCalcoloFormaturaWA[CalFor].TipoElementoDep[i] := LASTRA;//Settiamo tutte lastre!!
				ELSE
					TFCalcoloFormaturaWA[CalFor].TipoElementoDep[i] := TERMINATORE;//Settiamo il resto come terminatore
				END_IF
			END_FOR
		ELSE
			//FOR i := 1 TO HMI_Forming_NumeroElementiDaDepositare DO//BY (Request_WorkOrder.LayerSequence+1) DO		  
			FOR i := 1 TO HMI_Forming_NumeroElementiDaDepositare DO//BY (Request_WorkOrder.LayerSequence+1) DO
				// Pasaje Estructura dimensiones posicion piking
				TFCalcoloFormaturaWA[CalFor].Materiale[i].DimensionPiezasLadoALadoB := 
													HMi_DimensionesPiezasWorkAreaDeposito[i];
				IF i MOD 2 = 1 THEN// i <= HMI_Forming_NumeroElementiDaDepositare THEN 
					
					TFCalcoloFormaturaWA[CalFor].TipoElementoDep[i] := LASTRA;//Settiamo tipo lastre!!
				ELSE
					TFCalcoloFormaturaWA[CalFor].TipoElementoDep[i] := FALDA;//Settiamo tipoi falda!
				END_IF
					TFCalcoloFormaturaWA[CalFor].TipoElementoDep[i+1] := TERMINATORE;//Settiamo il resto come terminatore
			END_FOR
		END_IF	
		TFCalcoloFormaturaWA[CalFor].Materiale[e_Tipo_Elemento_Da_Lavorare.LASTRA]		:= HMI_Forming_LastraDaDepositare; 
		TFCalcoloFormaturaWA[CalFor].Materiale[e_Tipo_Elemento_Da_Lavorare.FALDA]		:= FaldaDaDepositare;
		TFCalcoloFormaturaWA[CalFor].Materiale[e_Tipo_Elemento_Da_Lavorare.QUADROTTA]	:= HMI_Forming_LastraDaDepositare;
		TFCalcoloFormaturaWA[CalFor].Supporto											:= HMI_Forming_Supporto;	//Assegno la tipologia di supporto
		
		TFCalcoloFormaturaWA[CalFor].DimensionesPiezasDifEsPiking     := HMi_DimensionesPiezasWorkAreaDeposito ;
		
	
		//CASE HMI_WorkAreaDataPicking[j].Typology OF //**Mod
	 
		CASE HMI_WorkAreaDataPicking[NumPostazioneDeposito].Typology OF //**Mod
			BUNDLE_VERT:
				TFCalcoloFormaturaWA[CalFor].TipoOrdinamento := 4;//Ordinamento di deposito òato 180°
			A_FRAME_VERT:
				TFCalcoloFormaturaWA[CalFor].TipoOrdinamento := 1;//Ordinamento di deposito, prima un lato poi l'altro	
				TFCalcoloFormaturaWA[CalFor].HabiCalTodasCordenadas := TRUE ;
			ELSE
				TFCalcoloFormaturaWA[CalFor].TipoOrdinamento := 2;//Ordinamento di deposito consecutivo	 
		END_CASE
			 
		TFCalcoloFormaturaWA[CalFor].CalcolaFormatura := TRUE; 		//Lancio esecuzione dei calcoli
				  
			IF HabilitapikingPruevas THEN 				
				TFCalcoloFormaturaWA[CalFor].CalculoEstacionPickinPiezasDiferentes := TRUE ;
	  		ELSE
				TFCalcoloFormaturaWA[CalFor].CalculoEstacionPickinPiezasDiferentes := FALSE ;		  
			END_IF
		MEMSET(ADR(HMI_Forming_FormaturaCalcolata),0,SIZEOF(HMI_Forming_FormaturaCalcolata));	//Pulisco la memoria di destinazione
		HMI_Forming_Attivazione[i] := FALSE;
		TFCalcoloFormaturaWA[CalFor].PulisciMemoria := FALSE;
		TFCalcoloFormaturaWA[CalFor]();
  
	 END_IF
			   
	IF (TFCalcoloFormaturaWA[CalFor].CalcolaFormaturaDone OR TFCalcoloFormaturaWA[CalFor].Errore > 0)AND NOT FormacionPikingCalculada THEN
		
		TFCalcoloFormaturaDaLista.CalcolaFormatura := FALSE;
		Formacion_De_listaOk[calfor] := TRUE ;
				IF TFCalcoloFormaturaWA[CalFor].Errore = 0 THEN
					IDFormatura 								:= IDFormatura+1;
					GUIDFormatura 								:= STRING_TO_UINT(concat(UINT_TO_STRING(NUMERO_MACCHINA),UINT_TO_STRING(IDFormatura)));
					HMI_Forming_GUID 							:= GUIDFormatura;
					HMI_Forming_FormaturaCalcolata 				:= TFCalcoloFormaturaWA[CalFor].FormingSlab;
					HMI_Forming_FormaturaAttivataWa[CalFor] 	:= TRUE ;

		  
					FormaturaWa[CalFor]							:= FormingEmpty;
					FormaturaWa[CalFor]	 						:= TFCalcoloFormaturaWA[CalFor].FormingSlab;
					FormaturaWa[CalFor].Enable 					:= 1;
					FormaturaWa[CalFor].Code 					:= HMI_Forming_CodiciAbilitatiFormatura[CalFor].Code;
					FormaturaWa[CalFor].GUID					:= HMI_Forming_GUID;
					FormaturaWa[CalFor].Pallet					:= HMI_Forming_Supporto;
							  
					
					Forming[idxForm] 							:= FormingEmpty;	//Pulisco la memoria di destinazione
					Forming[idxForm] 							:= TFCalcoloFormaturaWA[CalFor].FormingSlab;
					Forming[idxForm].Enable 						:= 1;
					Forming[idxForm].Code 						:= HMI_Forming_CodiciAbilitatiFormatura[CalFor].Code;
					Forming[idxForm].GUID						:= HMI_Forming_GUID;
					Forming[idxForm].Pallet						:= HMI_Forming_Supporto;
					HMI_Forming_IndiceFormaturaAttivata 		:= idxForm;
					HMI_Forming_FormaturaAttivata[CalFor] 		:= TRUE;
					HMI_ConfermaAttivazioneFormatura[CalFor] 	:= TRUE;
					FormacionPikingCalculada					:= TRUE ;
					//Valorizzo la struttura del WAPL per ogni elemento da elaborare
					FOR jj := 1 TO MAXELEMENTLIST DO
						IF jj < ElementiElaborati[IdxLista] THEN
							WorkAreaProductionList[CalFor].PElementList[jj].PElement 		:= TFCalcoloFormaturaWA[CalFor].FormingSlab.PElement[jj];	
							WorkAreaProductionList[CalFor].PElementList[jj].Stato			:= ELEMENTO_DA_ELABORARE;
						
							IF Picking.HMI_PareggiaturaLastraAbilitata THEN
								WorkAreaProductionList[CalFor].PElementList[jj].Pareggiatura := PAREGGIATURA_DA_ESEGUIRE;
							ELSE
								WorkAreaProductionList[CalFor].PElementList[jj].Pareggiatura := PAREGGIATURA_DISABILITATA;
							END_IF
						ELSE
							WorkAreaProductionList[CalFor].PElementList[jj].Stato			:= ELEMENTO_NOT_DEFINED;
						END_IF
					END_FOR
				ELSE
					HMI_Forming_ErroreCalcoli := TFCalcoloFormaturaWA[CalFor].Errore;
				END_IF
				HMI_Forming_Attivazione[idxForm] := FALSE;
			END_IF		  
	(* Metto in stato di esecuzione il nuovo W.O. se tutto si è attivato *)
		IF HMI_Forming_FormaturaAttivata[CalFor] THEN

			ActualPickingListFromHMI[idxForm].State := e_StatoWorkOrder.DA_ESEGUIRE;
			//Azzero le liste per le postazioni dove non avviene la pallettizzazione
			FOR i:= Iforstart TO Iforend DO		 
				WorkAreaProductionList[i].Stato := e_Stato_ListaDiProduzione.LISTA_PROD_ASSENTE;
			END_FOR
			//WorkAreaProductionList[NumPostazioneDeposito].Support := Forming[idxForm].Pallet;
			WorkAreaProductionList[CalFor].Stato 								:= LISTA_PROD_DA_ESEGUIRE;
			WorkAreaProductionList[CalFor].NumeroListaAssociata 				:= idxForm;
			WorkAreaState[CalFor].F 											:= idxForm;
			Picking.Cmd_CalcolaLista[IdxLista] 									:= FALSE;
			HMI_Forming_FormaturaAttivata[IdxLista] 							:= FALSE;
			
		END_IF	  
END_IF 
		  
					
							  
										
												  
IF HMI_Forming_FormaturaAttivataWa[NumPostazioneDeposito] AND NOT FormacionesCalculadas 	   THEN
		idxForm:= IdxLista;		  
		FOR CalFor := Iforstart TO Iforend DO
				
				IF CalFor <> NumPostazioneDeposito AND HMI_NumeroPezziPresentiPostazione[CalFor] > 0 AND HMI_WorkAreaDataPicking[CalFor].NumElementiDaLavorare <> 0 AND NOT FormacionesCalculadas  THEN // calcula la formacion para la estacion de piking
					MEMSET(destAddr := ADR(TFCalcoloFormaturaWA[CalFor]),fillByte := 0 , n := SIZEOF(TFCalcoloFormaturaWA[CalFor]));
					TFCalcoloFormaturaWA[CalFor].PulisciMemoria 			:= TRUE ; 
					TFCalcoloFormaturaWA[CalFor]();	
		 				IF TFCalcoloFormaturaWA[CalFor].PulisciMemoriaDone THEN		
							FOR i:= 1 TO MAXFORMINGSLAB DO
								IF i <= 40 THEN
								//IF i <= HMI_Forming_NumeroElementiDaDepositare THEN
									TFCalcoloFormaturaWA[CalFor].TipoElementoDep[i] := LASTRA;//Settiamo tutte lastre!!
								ELSE
									TFCalcoloFormaturaWA[CalFor].TipoElementoDep[i] := TERMINATORE;//Settiamo il resto come terminatore
								END_IF
							END_FOR
						TFCalcoloFormaturaWA[CalFor].Materiale[e_Tipo_Elemento_Da_Lavorare.LASTRA].XDim				:= RequestPickingListFromHMIWorkArea[CalFor].SlabDimension.XDim; 
						TFCalcoloFormaturaWA[CalFor].Materiale[e_Tipo_Elemento_Da_Lavorare.LASTRA].YDim				:= RequestPickingListFromHMIWorkArea[CalFor].SlabDimension.YDim; 
						TFCalcoloFormaturaWA[CalFor].Materiale[e_Tipo_Elemento_Da_Lavorare.LASTRA].ZDim				:= RequestPickingListFromHMIWorkArea[CalFor].SlabDimension.ZDim; 
						TFCalcoloFormaturaWA[CalFor].Supporto.Code													:= WorkAreaState[CalFor].Supporto.Code ;
						TFCalcoloFormaturaWA[CalFor].Supporto.XDim													:= WorkAreaState[CalFor].Supporto.XDim;
						TFCalcoloFormaturaWA[CalFor].Supporto.YDim													:= WorkAreaState[CalFor].Supporto.YDim ;
						TFCalcoloFormaturaWA[CalFor].Supporto.ZDim													:= WorkAreaState[CalFor].Supporto.ZDim;
						TFCalcoloFormaturaWA[CalFor].Supporto.DimBaseUtile											:= WorkAreaState[CalFor].Supporto.DimBaseUtile;
						TFCalcoloFormaturaWA[CalFor].Supporto.DimVertice 											:= WorkAreaState[CalFor].Supporto.DimVertice ;
						TFCalcoloFormaturaWA[CalFor].Supporto.HMAX 													:= WorkAreaState[CalFor].Supporto.HMAX;
							CASE  WorkAreaState[calfor].Supporto.Tipologia OF
								LEGNO_PIANO :
									HMI_Formatura.HMI_Forming_Supporto.Tipologia		:= e_Tipo_Pallet.CASSA_STANDARD;
												;
								TELAIO_PIANO : 
									HMI_Formatura.HMI_Forming_Supporto.Tipologia		:= e_Tipo_Pallet.CASSA_STANDARD;	 
												   
												;
								BUNDLE:
									TFCalcoloFormaturaWA[CalFor].Supporto.YDim											:= WorkAreaState[CalFor].Supporto.YDim*2;
									TFCalcoloFormaturaWA[CalFor].Supporto.DimVertice 									:= WorkAreaState[CalFor].Supporto.DimVertice*2;
									TFCalcoloFormaturaWA[CalFor].Supporto.TipoPianoAppoggio 							:= 1;
									TFCalcoloFormaturaWA[CalFor].Supporto.AltezzaDenteRitenuta							:= 15;
									TFCalcoloFormaturaWA[CalFor].Supporto.ZDim_Ext1        								:= TFCalcoloFormaturaWA[CalFor].Supporto.ZDim + TFCalcoloFormaturaWA[CalFor].Supporto.AltezzaDenteRitenuta;
									TFCalcoloFormaturaWA[CalFor].Supporto.Tipologia 									:= BUNDLE;
									TFCalcoloFormaturaWA[CalFor].Supporto.LatoDeposito 									:= 180;
									TFCalcoloFormaturaWA[CalFor].TipoOrdinamento										:= 4;	//Ordinamento di deposito, prima un lato poi l'altro
									
								A_FRAME_VERT:		  
									TFCalcoloFormaturaWA[CalFor].HabiCalTodasCordenadas 								:= TRUE ;
									TFCalcoloFormaturaWA[CalFor].Supporto.TipoPianoAppoggio 							:= 1;
									TFCalcoloFormaturaWA[CalFor].Supporto.AltezzaDenteRitenuta							:= 13;
									TFCalcoloFormaturaWA[CalFor].Supporto.ZDim_Ext1        								:= TFCalcoloFormaturaWA[CalFor].Supporto.ZDim + TFCalcoloFormaturaWA[CalFor].Supporto.AltezzaDenteRitenuta;
									TFCalcoloFormaturaWA[CalFor].Supporto.Tipologia 									:= CAVALLETTO;
									TFCalcoloFormaturaWA[CalFor].Supporto.LatoDeposito 									:= 0;
									TFCalcoloFormaturaWA[CalFor].TipoOrdinamento										:= 1;	//Ordinamento di deposito, prima un lato poi l'altro
									 
							END_CASE
							TFCalcoloFormaturaWA[CalFor].CalcolaFormatura 				:= TRUE;//Lancio esecuzione dei calcoli
							MEMSET(ADR(FormaturaWA[CalFor]),0,SIZEOF(FormaturaWA[CalFor]));	//Pulisco la memoria di destinazione
							TFCalcoloFormaturaWA[CalFor].PulisciMemoria 				:= FALSE;
							TFCalcoloFormaturaWA[CalFor]() ;
					END_IF
									
							
					 IF (TFCalcoloFormaturaWA[CalFor].CalcolaFormaturaDone OR TFCalcoloFormaturaWA[CalFor].Errore > 0) THEN
							
						TFCalcoloFormaturaWA[CalFor].CalcolaFormatura := FALSE;
						TFFormacionCavalleteCalculada := TFCalcoloFormaturaWA[CalFor] ;
						FormaturaWa[CalFor] := TFCalcoloFormaturaWA[CalFor].FormingSlab;
							//CalcolaFormingRT[IdxLista] := TRUE ; // modificacion probar
							IF TFCalcoloFormaturaRT[CalFor].Errore = 0 THEN
								HMI_Forming_FormaturaAttivataWa[CalFor] := TRUE ;
								IF  calfor = Iforend    THEN 
									FormacionesCalculadas := TRUE ;		  
								END_IF		  
							ELSE
								HMI_Forming_ErroreCalculos[CalFor] := TRUE ; 
							END_IF
					END_IF
								 
				 
	
			END_IF
		IF  calfor = Iforend  AND NOT FormacionesCalculadas  THEN 
			FormacionesCalculadas := TRUE ;	
			EXIT ;	  
		END_IF		  			  
	END_FOR
END_IF 															
																	  
{endregion}
	 

		






END_IF	
		
END_FOR	 
	 

	HMI_WorkAreaDataPicking_1_8 := ActualPickingListFromHMI[1].State >= 1;//Ordine postazioni 1..8 in lavoro
	HMI_WorkAreaDataPicking_1_4 := (ActualPickingListFromHMI[2].State >= 1);//Ordine postazioni 1..4 in lavoro
	HMI_WorkAreaDataPicking_5_8 := (ActualPickingListFromHMI[3].State >= 1);//Ordine postazioni 5..8 in lavoro


							  
								   
{endregion}
END_ACTION

ACTION _11_CalcolaListaProduzioneNew1:
{region "Gestione zona GLOBALE - Postazioni da 1 a 8"}


//#############################################################################################################



	  
	  

FOR LoopLista := 1 TO 3 DO
	IdxLista := LoopLista;		 
	 // IdxLista := 2;		  
	CASE IdxLista OF	 
		1: Iforstart := 1; Iforend := MAXAREAPRESENT;
		2: Iforstart := 1; Iforend := 4;
		3: Iforstart := 5; Iforend := MAXAREAPRESENT;
	END_CASE	 
	IF MachinePalletizer_TF.IN.Mode.Man AND
		(MachinePalletizer_TF.CmdExe.Code = CmdNOP OR MachinePalletizer_TF.CmdExe.Code = CmdMAN) THEN
			 
				  
					   
							
{region "Reset Litas"}
//--------------------------------------------------------
			//AZZERAMENTO (Reset) lista di picking	
//--------------------------------------------------------		 
			IF Cmd_AzzeraLista[IdxLista] THEN
				IF Prueva THEN
					MissionClr := ADR(Mission) ;
	 				MEMSET(destAddr := ADR(MissionClr^),fillByte := 0 , n := SIZEOF(MissionClr^));
				END_IF
					ClrEstructura := ADR(PosCavalleteOrdenPikin) ;
					MEMSET(destAddr := ADR(ClrEstructura^),fillByte := 0 , n := SIZEOF(ClrEstructura^));	  
					NuEstacionesPiking := 0 ;	  
					NuEstacionPiking   := 0 ;
					NuPosGuiroPiking := 0;
					PosFinOrdenPikingCaballete := 0 ;
					
					MultiplesCavalletesReceta := FALSE ;
					CoordenadaPasillo0_Y := 0 ;
					CoordenadaPasillo180_Y := 0 ;
					
				
				//FOR i:= 1 TO 3 DO
						//CalcolaFormingRT2[i] := FALSE ;
					CalcolaFormingRT[IdxLista] := FALSE ;
					CalcolaFormingRT2[IdxLista] := FALSE ;	 
						//#Añadido 4_7_2025########################
					Formacion_bandelCalOk[IdxLista]			:= FALSE ;
					Formacion_FrameCalOk[IdxLista]			:= FALSE ;
					Formacion_De_listaOk[IdxLista]			:= FALSE ;
					FormaturaAFRAMERT[IdxLista]		   	:=	FormingEmpty;
					FormaturaBundleRT[IdxLista]	 		:=	FormingEmpty;
							  
					MEMSET(destAddr := ADR(TFFormacionBandelCalculada),fillByte := 0 , n := SIZEOF(TFFormacionBandelCalculada));
					MEMSET(destAddr := ADR(TFFormacionCavalleteCalculada),fillByte := 0 , n := SIZEOF(TFFormacionCavalleteCalculada));
					MEMSET(destAddr := ADR(TFCalcoloFormaturaWA),fillByte := 0 , n := SIZEOF(TFCalcoloFormaturaWA));
					
		  
				//Añadido 4_7_2025##########################
						
				// END_FOR
				ActualPickingListFromHMI[IdxLista].State := e_StatoWorkOrder.NON_ESEGUITO;
				HMI_NumeroLastreDepOrdineAttuale[IdxLista] := 0; 
				//Disattivazione formatura
				Forming[1] := FormingEmpty;	//Pulisco la formatura selezionata e di consegenza la disattivo
				Forming[2] := FormingEmpty;	//Pulisco la formatura selezionata e di consegenza la disattivo
				Forming[3] := FormingEmpty;	//Pulisco la formatura selezionata e di consegenza la disattivo
				Forming[4] := FormingEmpty;	//Pulisco la formatura selezionata e di consegenza la disattivo
				ActualPickingListFromHMI[IdxLista].State := e_StatoWorkOrder.NON_ESEGUITO;
				Cmd_AttivaLista[IdxLista] := FALSE;
				HMI_Forming_NumeroElementiDaDepositare := 0;
 				RequestPickingListFromHMI[IdxLista].SlabNumber :=0;
	 
				//Azzero le liste per le postazioni dove non avviene la pallettizzazione
				FOR i:= Iforstart TO Iforend DO	
					TFClearWorkAreaArray(ADR(Workarea),ADR(WorkAreaState),k:=i);
					HMI_WorkAreaDataPicking[i].Destinazione := FALSE;
					HMI_WorkAreaDataPicking[i].NumElementiDaLavorare := 0;
					WorkAreaState[i].P 			:= 1;
					WorkAreaProductionList[i] 	:= ListaEmpty;
					WorkAreaOffset[i].Y 		:= 0;
					//HMI_NumeroPezziPresentiPostazione[i] 	:= 0; // Quitado Para No resetear posiciones
					NumeroPezziPresentiPostazioneStart[i] 	:= 0;
					WorkAreaProductionList[i].Stato 		:= e_Stato_ListaDiProduzione.LISTA_PROD_ASSENTE;	 
				END_FOR			  
				ActualPickingListFromHMI[IdxLista].SlabNumber 		  			:= 0;
				ActualPickingListFromHMI[IdxLista].SlabDimension.XDim 			:= 0;
				ActualPickingListFromHMI[IdxLista].SlabDimension.YDim 			:= 0;
				ActualPickingListFromHMI[IdxLista].SlabDimension.ZDim 			:= 0;
				ActualPickingListFromHMI[IdxLista].SupportPianoLegno 			:= SupportDataEmpty;
				ActualPickingListFromHMI[IdxLista].SupportPianoFerro 			:= SupportDataEmpty;
				ActualPickingListFromHMI[IdxLista].SupportVertBundle 			:= SupportDataEmpty;
				ActualPickingListFromHMI[IdxLista].SupportVertCav 			 	:= SupportDataEmpty;
				
				HMI_ErroreCalcoloLista 		:= 0;
				Cmd_CalcolaLista[IdxLista] 	:= FALSE;
				HMI_Forming_Attivazione[IdxLista] 	:= FALSE;//attivo nuova formatura
				Cmd_AzzeraLista[IdxLista] := FALSE;
				//Ack 
				//IF HMI_ErrAckCalcolaFormatura THEN
					HMI_Forming_ErroreCalcoli := 0;
					HMI_ErrAckCalcolaFormatura := FALSE;
					FOR i:= 1 TO MAXFORMING DO
						HMI_ConfermaAttivazioneFormatura[i] := FALSE;
						HMI_Forming_FormaturaAttivata[i] := FALSE;
					END_FOR
				//END_IF
				CalcolaFormaturaTrig := FALSE;
			END_IF

{endregion}

//--------------------------------------------------------
		// COMANDO ATTIVAZIONE  lista di picking	
//--------------------------------------------------------		 		  
			//Se non ho una Destinazione impostata, Num.pezzi impostato, o Num.pezzi richiesto...
			//	Resetto il comando		
					IF Cmd_AttivaLista[1] = TRUE  THEN
							FOR uu := Iforstart TO Iforend DO
							 	IF	HMI_WorkAreaDataPicking[uu].Typology = CAVALLETTO THEN 
									CASE HMI_WorkAreaDataPicking[uu].TipoTrabajoLado_Cavallete OF 
	 									0:
											HMI_NumeroPezziPresentiPostazione[uu] := HMI_NumeroPezziPresentiCavallete[uu].HMI_NumeroPezziPresentiPostazione_A_Cavaleto +
												 HMI_NumeroPezziPresentiCavallete[uu].HMI_NumeroPezziPresentiPostazione_B_Cavaleto ;
										1:
											HMI_NumeroPezziPresentiPostazione[uu] := HMI_NumeroPezziPresentiCavallete[uu].HMI_NumeroPezziPresentiPostazione_A_Cavaleto ;									 ;
											 
										2:	
		   									HMI_NumeroPezziPresentiPostazione[uu] := HMI_NumeroPezziPresentiCavallete[uu].HMI_NumeroPezziPresentiPostazione_B_Cavaleto ;
												 
									END_CASE
								END_IF 	 
							END_FOR
								  
						IF 	(HMI_WorkAreaDataPicking[1].Destinazione =0 AND 
							HMI_WorkAreaDataPicking[2].Destinazione =0 AND
							HMI_WorkAreaDataPicking[3].Destinazione =0 AND 
							HMI_WorkAreaDataPicking[4].Destinazione =0 AND	 
							HMI_WorkAreaDataPicking[5].Destinazione =0 AND 
							HMI_WorkAreaDataPicking[6].Destinazione =0 AND
							HMI_WorkAreaDataPicking[7].Destinazione =0 AND 
							HMI_WorkAreaDataPicking[8].Destinazione =0)							 
							OR
							(HMI_NumeroPezziPresentiPostazione[1] =0 AND 
							HMI_NumeroPezziPresentiPostazione[2] =0 AND
							HMI_NumeroPezziPresentiPostazione[3] =0 AND 
							HMI_NumeroPezziPresentiPostazione[4] =0 AND
							HMI_NumeroPezziPresentiPostazione[5] =0 AND 
	 						HMI_NumeroPezziPresentiPostazione[6] =0 AND
							HMI_NumeroPezziPresentiPostazione[7] =0 AND 
							HMI_NumeroPezziPresentiPostazione[8] =0)
							OR	 	 
							RequestPickingListFromHMI[1].SlabNumber = 0	 
						THEN
							Cmd_AttivaLista[1] := FALSE;
						 END_IF
					END_IF		  
					IF Cmd_AttivaLista[2] = TRUE  THEN
						IF 	(HMI_WorkAreaDataPicking[1].Destinazione =0 AND 
							HMI_WorkAreaDataPicking[2].Destinazione =0 AND
							HMI_WorkAreaDataPicking[3].Destinazione =0 AND 
							HMI_WorkAreaDataPicking[4].Destinazione =0)
							OR
							(HMI_NumeroPezziPresentiPostazione[1] =0 AND 
							HMI_NumeroPezziPresentiPostazione[2] =0 AND
							HMI_NumeroPezziPresentiPostazione[3] =0 AND 
							HMI_NumeroPezziPresentiPostazione[4] =0)
							OR	 
							RequestPickingListFromHMI[2].SlabNumber = 0	 	 
						THEN
							Cmd_AttivaLista[2] := FALSE;
						 END_IF
					END_IF		
					IF Cmd_AttivaLista[3] = TRUE  THEN
						IF 	(HMI_WorkAreaDataPicking[5].Destinazione =0 AND 
							HMI_WorkAreaDataPicking[6].Destinazione =0 AND
							HMI_WorkAreaDataPicking[7].Destinazione =0 AND 
							HMI_WorkAreaDataPicking[8].Destinazione =0)
							OR
							(HMI_NumeroPezziPresentiPostazione[5] =0 AND 
							HMI_NumeroPezziPresentiPostazione[6] =0 AND
							HMI_NumeroPezziPresentiPostazione[7] =0 AND 
							HMI_NumeroPezziPresentiPostazione[8] =0)
							OR	 	 
							RequestPickingListFromHMI[3].SlabNumber = 0	 	 
						THEN
							Cmd_AttivaLista[3] := FALSE;
						 END_IF
					END_IF		
{Region "Prmer Bucle cuenta las piezas a coger y rellena el workareastate Con el Tipo Palet"}

			// COMANDO ATTIVAZIONE  lista di picking	
		    IF Cmd_AttivaLista[IdxLista] AND ActualPickingListFromHMI[IdxLista].State <> e_StatoWorkOrder.IN_ESECUZIONE THEN
				ElementiDaDepositare[IdxLista]   :=0;
				HMI_ErroreCalcoloLista := 0;
				HMI_NumeroLastreDepOrdineAttuale[IdxLista] := 0;
				FOR i:= Iforstart TO Iforend DO	
					//HMI_WorkAreaDataPicking[i].Destinazione := FALSE;
					//HMI_WorkAreaDataPicking[i].NumElementiDaLavorare := 0;
					WorkAreaState[i].P := 1;
					WorkAreaProductionList[i] := ListaEmpty;
				END_FOR	 
				
				FOR i:= Iforstart TO Iforend DO	
					IF NOT HMI_WorkAreaDataPicking[i].Destinazione THEN
						ElementiDaDepositare[IdxLista] := ElementiDaDepositare[IdxLista] + HMI_WorkAreaDataPicking[i].NumElementiDaLavorare;
						WorkAreaState[i].P := HMI_WorkAreaDataPicking[i].NumElementiDaLavorare +1;
					//#####################################################################################
							FOR InPiezasPos := 1 TO HMI_NumeroPezziPresentiPostazione[i] + 1 DO
								WorkAreaProductionList[i].PElementList[InPiezasPos].PElement.SlabDimension :=
																	 RequestPickingListFromHMIWorkArea[i].SlabDimension ;
								WorkAreaProductionList[i].PElementList[InPiezasPos].PElement.Typology := LASTRA ;
											   
							END_FOR
					//#################################################################################################	
						CASE HMI_WorkAreaDataPicking[i].Typology OF
							LEGNO_PIANO,TELAIO_PIANO:
								WorkareaState[i].Supporto.Tipologia := e_Tipo_Pallet.CASSA_STANDARD;
							A_FRAME_VERT:	
								WorkareaState[i].Supporto.Tipologia := e_Tipo_Pallet.CAVALLETTO;
								
